LIN {X 0,Y 559.905,Z 784.141,A -85,B 0,C 180,E1 26458.055,E2 26458.055} C_VEL
LIN {X 0,Y 559.916,Z 781.549,A -85,B 0,C 180,E1 26456.109,E2 26456.109} C_VEL
LIN {X 0,Y 559.927,Z 777.44,A -85,B 0,C 180,E1 26454.261,E2 26454.261} C_VEL
LIN {X 0,Y 559.97,Z 771.528,A -85,B 0,C 180,E1 26452.407,E2 26452.407} C_VEL
LIN {X 0,Y 560.042,Z 763.726,A -85,B 0,C 180,E1 26450.546,E2 26450.546} C_VEL
LIN {X 0,Y 560.172,Z 754.398,A -85,B 0,C 180,E1 26448.781,E2 26448.781} C_VEL
LIN {X 0,Y 560.352,Z 743.578,A -85,B 0,C 180,E1 26447.112,E2 26447.112} C_VEL
LIN {X 0,Y 560.59,Z 731.187,A -85,B 0,C 180,E1 26445.54,E2 26445.54} C_VEL
LIN {X 0,Y 560.897,Z 717.221,A -85,B 0,C 180,E1 26444.066,E2 26444.066} C_VEL
LIN {X 0,Y 561.232,Z 702.873,A -85,B 0,C 180,E1 26442.798,E2 26442.798} C_VEL
LIN {X 0,Y 561.61,Z 686.59,A -85,B 0,C 180,E1 26441.61,E2 26441.61} C_VEL
LIN {X 0,Y 561.993,Z 668.948,A -85,B 0,C 180,E1 26440.567,E2 26440.567} C_VEL
LIN {X 0,Y 562.027,Z 667.326,A -85,B 0,C 180,E1 26440.483,E2 26440.483} C_VEL
LIN {X 0,Y 561.268,Z 660.484,A -85,B 0,C 180,E1 26440.115,E2 26440.115} C_VEL
LIN {X 0,Y 555.955,Z 643.327,A -85,B 0,C 180,E1 26439.189,E2 26439.189} C_VEL
LIN {X 0,Y 555.08,Z 636.153,A -85,B 0,C 180,E1 26438.903,E2 26438.903} C_VEL
LIN {X 0,Y 555.365,Z 617.419,A -85,B 0,C 180,E1 26438.404,E2 26438.404} C_VEL
LIN {X 0,Y 555.537,Z 595.534,A -85,B 0,C 180,E1 26438.046,E2 26438.046} C_VEL
LIN {X 0,Y 556.229,Z 411.604,A -85,B 0,C 180,E1 26435.545,E2 26435.545} C_VEL
LIN {X 0,Y 554.815,Z 403.726,A -85,B 0,C 180,E1 26435.342,E2 26435.342} C_VEL
LIN {X 0,Y 555.413,Z 371.536,A -85,B 0,C 180,E1 26432.441,E2 26432.441} C_VEL
LIN {X 0,Y 555.301,Z 368.267,A -85,B 0,C 180,E1 26432.139,E2 26432.139} C_VEL
LIN {X 0,Y 552.299,Z 358.003,A -85,B 0,C 180,E1 26431.014,E2 26431.014} C_VEL
LIN {X 0,Y 552.268,Z 358.001,A -85,B 0,C 180,E1 26427.718,E2 26427.718} C_VEL
LIN {X 0,Y 552.338,Z 357.999,A -85,B 0,C 180,E1 26424.549,E2 26424.549} C_VEL
LIN {X 0,Y 552.269,Z 358,A -85,B 0,C 180,E1 26421.346,E2 26421.346} C_VEL
LIN {X 0,Y 552.297,Z 358.001,A -85,B 0,C 180,E1 26418.079,E2 26418.079} C_VEL
LIN {X 0,Y 552.288,Z 357.999,A -85,B 0,C 180,E1 26414.938,E2 26414.938} C_VEL
LIN {X 0,Y 552.269,Z 357.999,A -85,B 0,C 180,E1 26411.607,E2 26411.607} C_VEL
LIN {X 0,Y 552.329,Z 357.999,A -85,B 0,C 180,E1 26408.516,E2 26408.516} C_VEL
LIN {X 0,Y 552.266,Z 358,A -85,B 0,C 180,E1 26405.262,E2 26405.262} C_VEL
LIN {X 0,Y 552.312,Z 358,A -85,B 0,C 180,E1 26402.034,E2 26402.034} C_VEL
LIN {X 0,Y 552.27,Z 357.999,A -85,B 0,C 180,E1 26399.02,E2 26399.02} C_VEL
LIN {X 0,Y 552.278,Z 358,A -85,B 0,C 180,E1 26395.631,E2 26395.631} C_VEL
LIN {X 0,Y 552.299,Z 357.998,A -85,B 0,C 180,E1 26392.569,E2 26392.569} C_VEL
LIN {X 0,Y 552.267,Z 358,A -85,B 0,C 180,E1 26389.349,E2 26389.349} C_VEL
LIN {X 0,Y 552.335,Z 357.998,A -85,B 0,C 180,E1 26386.187,E2 26386.187} C_VEL
LIN {X 0,Y 552.263,Z 357.998,A -85,B 0,C 180,E1 26383.08,E2 26383.08} C_VEL
LIN {X 0,Y 552.322,Z 357.999,A -85,B 0,C 180,E1 26379.903,E2 26379.903} C_VEL
LIN {X 0,Y 552.271,Z 357.999,A -85,B 0,C 180,E1 26376.758,E2 26376.758} C_VEL
LIN {X 0,Y 552.272,Z 357.999,A -85,B 0,C 180,E1 26373.321,E2 26373.321} C_VEL
LIN {X 0,Y 552.311,Z 357.999,A -85,B 0,C 180,E1 26370.207,E2 26370.207} C_VEL
LIN {X 0,Y 552.263,Z 357.998,A -85,B 0,C 180,E1 26366.99,E2 26366.99} C_VEL
LIN {X 0,Y 552.327,Z 357.999,A -85,B 0,C 180,E1 26363.764,E2 26363.764} C_VEL
LIN {X 0,Y 552.268,Z 357.999,A -85,B 0,C 180,E1 26360.622,E2 26360.622} C_VEL
LIN {X 0,Y 552.277,Z 358,A -85,B 0,C 180,E1 26357.24,E2 26357.24} C_VEL
LIN {X 0,Y 552.287,Z 358,A -85,B 0,C 180,E1 26354.243,E2 26354.243} C_VEL
LIN {X 0,Y 552.265,Z 358,A -85,B 0,C 180,E1 26350.921,E2 26350.921} C_VEL
LIN {X 0,Y 552.339,Z 357.999,A -85,B 0,C 180,E1 26347.769,E2 26347.769} C_VEL
LIN {X 0,Y 552.263,Z 358,A -85,B 0,C 180,E1 26344.59,E2 26344.59} C_VEL
LIN {X 0,Y 552.302,Z 358,A -85,B 0,C 180,E1 26341.331,E2 26341.331} C_VEL
LIN {X 0,Y 552.27,Z 358,A -85,B 0,C 180,E1 26338.312,E2 26338.312} C_VEL
LIN {X 0,Y 552.267,Z 358.001,A -85,B 0,C 180,E1 26334.849,E2 26334.849} C_VEL
LIN {X 0,Y 552.334,Z 358.001,A -85,B 0,C 180,E1 26331.613,E2 26331.613} C_VEL
LIN {X 0,Y 552.262,Z 358,A -85,B 0,C 180,E1 26328.394,E2 26328.394} C_VEL
LIN {X 0,Y 552.292,Z 358.001,A -85,B 0,C 180,E1 26325.085,E2 26325.085} C_VEL
LIN {X 0,Y 552.275,Z 358,A -85,B 0,C 180,E1 26322.057,E2 26322.057} C_VEL
LIN {X 0,Y 552.266,Z 358.001,A -85,B 0,C 180,E1 26318.654,E2 26318.654} C_VEL
LIN {X 0,Y 552.33,Z 358.001,A -85,B 0,C 180,E1 26315.45,E2 26315.45} C_VEL
LIN {X 0,Y 552.26,Z 358.003,A -85,B 0,C 180,E1 26312.274,E2 26312.274} C_VEL
LIN {X 0,Y 552.306,Z 358.003,A -85,B 0,C 180,E1 26309.024,E2 26309.024} C_VEL
LIN {X 0,Y 552.265,Z 358.028,A -85,B 0,C 180,E1 26308.41,E2 26308.41} C_VEL
LIN {X 0,Y 554.662,Z 367.675,A -85,B 0,C 180,E1 26307.134,E2 26307.134} C_VEL
LIN {X 0,Y 554.097,Z 397.179,A -85,B 0,C 180,E1 26303.728,E2 26303.728} C_VEL
LIN {X 0,Y 553.581,Z 425.304,A -85,B 0,C 180,E1 26300.512,E2 26300.512} C_VEL
LIN {X 0,Y 553.056,Z 456.362,A -85,B 0,C 180,E1 26297.03,E2 26297.03} C_VEL
LIN {X 0,Y 552.732,Z 481.06,A -85,B 0,C 180,E1 26294.338,E2 26294.338} C_VEL
LIN {X 0,Y 553.464,Z 488.754,A -85,B 0,C 180,E1 26294.218,E2 26294.218} C_VEL
LIN {X 0,Y 553.107,Z 591.575,A -85,B 0,C 180,E1 26292.854,E2 26292.854} C_VEL
LIN {X 0,Y 553.014,Z 606.185,A -85,B 0,C 180,E1 26292.489,E2 26292.489} C_VEL
LIN {X 0,Y 552.864,Z 619.873,A -85,B 0,C 180,E1 26291.946,E2 26291.946} C_VEL
LIN {X 0,Y 552.676,Z 631.744,A -85,B 0,C 180,E1 26291.319,E2 26291.319} C_VEL
LIN {X 0,Y 552.466,Z 644.76,A -85,B 0,C 180,E1 26290.427,E2 26290.427} C_VEL
LIN {X 0,Y 552.307,Z 655.904,A -85,B 0,C 180,E1 26289.43,E2 26289.43} C_VEL
LIN {X 0,Y 552.166,Z 665.819,A -85,B 0,C 180,E1 26288.33,E2 26288.33} C_VEL
LIN {X 0,Y 552.044,Z 675.086,A -85,B 0,C 180,E1 26287.003,E2 26287.003} C_VEL
LIN {X 0,Y 551.979,Z 681.519,A -85,B 0,C 180,E1 26285.822,E2 26285.822} C_VEL
LIN {X 0,Y 551.94,Z 687.227,A -85,B 0,C 180,E1 26284.468,E2 26284.468} C_VEL
LIN {X 0,Y 551.92,Z 691.681,A -85,B 0,C 180,E1 26282.908,E2 26282.908} C_VEL
LIN {X 0,Y 551.916,Z 693.98,A -85,B 0,C 180,E1 26281.557,E2 26281.557} C_VEL
LIN {X 0,Y 551.916,Z 694.996,A -85,B 0,C 180,E1 26280,E2 26280} C_VEL
LIN {X 0,Y 551.918,Z 694.092,A -85,B 0,C 180,E1 26278.443,E2 26278.443} C_VEL
LIN {X 0,Y 551.919,Z 691.869,A -85,B 0,C 180,E1 26277.093,E2 26277.093} C_VEL
LIN {X 0,Y 551.935,Z 687.911,A -85,B 0,C 180,E1 26275.637,E2 26275.637} C_VEL
LIN {X 0,Y 551.974,Z 681.957,A -85,B 0,C 180,E1 26274.178,E2 26274.178} C_VEL
LIN {X 0,Y 552.043,Z 675.194,A -85,B 0,C 180,E1 26272.926,E2 26272.926} C_VEL
LIN {X 0,Y 552.158,Z 666.551,A -85,B 0,C 180,E1 26271.671,E2 26271.671} C_VEL
LIN {X 0,Y 552.296,Z 656.805,A -85,B 0,C 180,E1 26270.57,E2 26270.57} C_VEL
LIN {X 0,Y 552.442,Z 647.08,A -85,B 0,C 180,E1 26269.678,E2 26269.678} C_VEL
LIN {X 0,Y 552.635,Z 634.983,A -85,B 0,C 180,E1 26268.785,E2 26268.785} C_VEL
LIN {X 0,Y 552.84,Z 621.669,A -85,B 0,C 180,E1 26268.049,E2 26268.049} C_VEL
LIN {X 0,Y 552.988,Z 609.624,A -85,B 0,C 180,E1 26267.546,E2 26267.546} C_VEL
LIN {X 0,Y 553.147,Z 595.043,A -85,B 0,C 180,E1 26267.121,E2 26267.121} C_VEL
LIN {X 0,Y 553.225,Z 571.612,A -85,B 0,C 180,E1 26266.771,E2 26266.771} C_VEL
LIN {X 0,Y 553.235,Z 484.541,A -85,B 0,C 180,E1 26265.631,E2 26265.631} C_VEL
LIN {X 0,Y 552.731,Z 480.548,A -85,B 0,C 180,E1 26265.544,E2 26265.544} C_VEL
LIN {X 0,Y 553.202,Z 451.312,A -85,B 0,C 180,E1 26262.271,E2 26262.271} C_VEL
LIN {X 0,Y 553.876,Z 420.903,A -85,B 0,C 180,E1 26258.781,E2 26258.781} C_VEL
LIN {X 0,Y 554.628,Z 391.683,A -85,B 0,C 180,E1 26255.39,E2 26255.39} C_VEL
LIN {X 0,Y 555.131,Z 368.311,A -85,B 0,C 180,E1 26252.618,E2 26252.618} C_VEL
LIN {X 0,Y 552.283,Z 358.006,A -85,B 0,C 180,E1 26251.153,E2 26251.153} C_VEL
LIN {X 0,Y 552.267,Z 358.004,A -85,B 0,C 180,E1 26247.841,E2 26247.841} C_VEL
LIN {X 0,Y 552.323,Z 358.001,A -85,B 0,C 180,E1 26244.727,E2 26244.727} C_VEL
LIN {X 0,Y 552.263,Z 358.003,A -85,B 0,C 180,E1 26241.611,E2 26241.611} C_VEL
LIN {X 0,Y 552.335,Z 358,A -85,B 0,C 180,E1 26238.506,E2 26238.506} C_VEL
LIN {X 0,Y 552.264,Z 358.002,A -85,B 0,C 180,E1 26235.359,E2 26235.359} C_VEL
LIN {X 0,Y 552.301,Z 358.003,A -85,B 0,C 180,E1 26232.077,E2 26232.077} C_VEL
LIN {X 0,Y 552.274,Z 358.002,A -85,B 0,C 180,E1 26229.043,E2 26229.043} C_VEL
LIN {X 0,Y 552.27,Z 358.005,A -85,B 0,C 180,E1 26225.621,E2 26225.621} C_VEL
LIN {X 0,Y 552.346,Z 358.153,A -85,B 0,C 180,E1 26222.461,E2 26222.461} C_VEL
LIN {X 0,Y 556.828,Z 371.461,A -85,B 0,C 180,E1 26221.141,E2 26221.141} C_VEL
LIN {X 0,Y 556.025,Z 413.458,A -85,B 0,C 180,E1 26218.049,E2 26218.049} C_VEL
LIN {X 0,Y 555.335,Z 457.917,A -85,B 0,C 180,E1 26214.917,E2 26214.917} C_VEL
LIN {X 0,Y 555.345,Z 463.245,A -85,B 0,C 180,E1 26214.568,E2 26214.568} C_VEL
LIN {X 0,Y 556.414,Z 472.063,A -85,B 0,C 180,E1 26214.395,E2 26214.395} C_VEL
LIN {X 0,Y 555.439,Z 672.312,A -85,B 0,C 180,E1 26211.656,E2 26211.656} C_VEL
LIN {X 0,Y 555.177,Z 691.233,A -85,B 0,C 180,E1 26211.202,E2 26211.202} C_VEL
LIN {X 0,Y 554.831,Z 709.39,A -85,B 0,C 180,E1 26210.574,E2 26210.574} C_VEL
LIN {X 0,Y 554.427,Z 727.031,A -85,B 0,C 180,E1 26209.764,E2 26209.764} C_VEL
LIN {X 0,Y 554.003,Z 743.688,A -85,B 0,C 180,E1 26208.799,E2 26208.799} C_VEL
LIN {X 0,Y 553.575,Z 759.623,A -85,B 0,C 180,E1 26207.664,E2 26207.664} C_VEL
LIN {X 0,Y 553.162,Z 774.553,A -85,B 0,C 180,E1 26206.378,E2 26206.378} C_VEL
LIN {X 0,Y 552.809,Z 788.017,A -85,B 0,C 180,E1 26204.99,E2 26204.99} C_VEL
LIN {X 0,Y 552.497,Z 800.914,A -85,B 0,C 180,E1 26203.394,E2 26203.394} C_VEL
LIN {X 0,Y 552.266,Z 812.229,A -85,B 0,C 180,E1 26201.699,E2 26201.699} C_VEL
LIN {X 0,Y 552.096,Z 822.169,A -85,B 0,C 180,E1 26199.871,E2 26199.871} C_VEL
LIN {X 0,Y 551.99,Z 830.178,A -85,B 0,C 180,E1 26198.018,E2 26198.018} C_VEL
LIN {X 0,Y 551.941,Z 836.414,A -85,B 0,C 180,E1 26196.136,E2 26196.136} C_VEL
LIN {X 0,Y 551.914,Z 840.877,A -85,B 0,C 180,E1 26194.26,E2 26194.26} C_VEL
LIN {X 0,Y 551.911,Z 843.792,A -85,B 0,C 180,E1 26192.284,E2 26192.284} C_VEL
LIN {X 0,Y 551.908,Z 844.94,A -85,B 0,C 180,E1 26190.311,E2 26190.311} C_VEL
LIN {X 0,Y 551.913,Z 844.416,A -85,B 0,C 180,E1 26188.443,E2 26188.443} C_VEL
LIN {X 0,Y 551.91,Z 842.163,A -85,B 0,C 180,E1 26186.469,E2 26186.469} C_VEL
LIN {X 0,Y 551.93,Z 838.35,A -85,B 0,C 180,E1 26184.595,E2 26184.595} C_VEL
LIN {X 0,Y 551.973,Z 832.818,A -85,B 0,C 180,E1 26182.715,E2 26182.715} C_VEL
LIN {X 0,Y 552.055,Z 825.427,A -85,B 0,C 180,E1 26180.829,E2 26180.829} C_VEL
LIN {X 0,Y 552.183,Z 816.517,A -85,B 0,C 180,E1 26179.04,E2 26179.04} C_VEL
LIN {X 0,Y 552.389,Z 805.985,A -85,B 0,C 180,E1 26177.323,E2 26177.323} C_VEL
LIN {X 0,Y 552.656,Z 794.351,A -85,B 0,C 180,E1 26175.756,E2 26175.756} C_VEL
LIN {X 0,Y 553.008,Z 780.575,A -85,B 0,C 180,E1 26174.21,E2 26174.21} C_VEL
LIN {X 0,Y 553.415,Z 765.602,A -85,B 0,C 180,E1 26172.819,E2 26172.819} C_VEL
LIN {X 0,Y 553.854,Z 749.432,A -85,B 0,C 180,E1 26171.583,E2 26171.583} C_VEL
LIN {X 0,Y 554.274,Z 733.051,A -85,B 0,C 180,E1 26170.56,E2 26170.56} C_VEL
LIN {X 0,Y 554.689,Z 715.808,A -85,B 0,C 180,E1 26169.696,E2 26169.696} C_VEL
LIN {X 0,Y 555.062,Z 697.521,A -85,B 0,C 180,E1 26168.994,E2 26168.994} C_VEL
LIN {X 0,Y 555.352,Z 678.843,A -85,B 0,C 180,E1 26168.48,E2 26168.48} C_VEL
LIN {X 0,Y 555.535,Z 658.475,A -85,B 0,C 180,E1 26168.131,E2 26168.131} C_VEL
LIN {X 0,Y 556.263,Z 469.166,A -85,B 0,C 180,E1 26165.558,E2 26165.558} C_VEL
LIN {X 0,Y 555.257,Z 462.604,A -85,B 0,C 180,E1 26165.417,E2 26165.417} C_VEL
LIN {X 0,Y 556.077,Z 416.365,A -85,B 0,C 180,E1 26162.128,E2 26162.128} C_VEL
LIN {X 0,Y 556.788,Z 373.888,A -85,B 0,C 180,E1 26159.037,E2 26159.037} C_VEL
LIN {X 0,Y 556.714,Z 371.068,A -85,B 0,C 180,E1 26158.815,E2 26158.815} C_VEL
LIN {X 0,Y 552.323,Z 357.992,A -85,B 0,C 180,E1 26157.521,E2 26157.521} C_VEL
LIN {X 0,Y 552.27,Z 358.001,A -85,B 0,C 180,E1 26154.38,E2 26154.38} C_VEL
LIN {X 0,Y 552.273,Z 358.001,A -85,B 0,C 180,E1 26150.947,E2 26150.947} C_VEL
LIN {X 0,Y 552.3,Z 358.002,A -85,B 0,C 180,E1 26147.923,E2 26147.923} C_VEL
LIN {X 0,Y 552.263,Z 358.001,A -85,B 0,C 180,E1 26144.641,E2 26144.641} C_VEL
LIN {X 0,Y 552.338,Z 358,A -85,B 0,C 180,E1 26141.458,E2 26141.458} C_VEL
LIN {X 0,Y 552.262,Z 358.002,A -85,B 0,C 180,E1 26138.377,E2 26138.377} C_VEL
LIN {X 0,Y 552.307,Z 358.003,A -85,B 0,C 180,E1 26135.148,E2 26135.148} C_VEL
LIN {X 0,Y 552.271,Z 358.005,A -85,B 0,C 180,E1 26132.037,E2 26132.037} C_VEL
LIN {X 0,Y 552.288,Z 358.066,A -85,B 0,C 180,E1 26128.808,E2 26128.808} C_VEL
LIN {X 0,Y 555.368,Z 369.2,A -85,B 0,C 180,E1 26127.652,E2 26127.652} C_VEL
LIN {X 0,Y 555.188,Z 387.302,A -85,B 0,C 180,E1 26126.067,E2 26126.067} C_VEL
LIN {X 0,Y 554.885,Z 404.57,A -85,B 0,C 180,E1 26124.525,E2 26124.525} C_VEL
LIN {X 0,Y 556.376,Z 413.773,A -85,B 0,C 180,E1 26124.328,E2 26124.328} C_VEL
LIN {X 0,Y 555.435,Z 612.55,A -85,B 0,C 180,E1 26121.607,E2 26121.607} C_VEL
LIN {X 0,Y 555.154,Z 632.028,A -85,B 0,C 180,E1 26121.134,E2 26121.134} C_VEL
LIN {X 0,Y 554.826,Z 649.668,A -85,B 0,C 180,E1 26120.518,E2 26120.518} C_VEL
LIN {X 0,Y 554.401,Z 668.293,A -85,B 0,C 180,E1 26119.655,E2 26119.655} C_VEL
LIN {X 0,Y 553.957,Z 685.572,A -85,B 0,C 180,E1 26118.63,E2 26118.63} C_VEL
LIN {X 0,Y 553.523,Z 701.786,A -85,B 0,C 180,E1 26117.449,E2 26117.449} C_VEL
LIN {X 0,Y 553.108,Z 716.635,A -85,B 0,C 180,E1 26116.13,E2 26116.13} C_VEL
LIN {X 0,Y 552.756,Z 730.434,A -85,B 0,C 180,E1 26114.669,E2 26114.669} C_VEL
LIN {X 0,Y 552.461,Z 742.929,A -85,B 0,C 180,E1 26113.075,E2 26113.075} C_VEL
LIN {X 0,Y 552.229,Z 753.85,A -85,B 0,C 180,E1 26111.382,E2 26111.382} C_VEL
LIN {X 0,Y 552.076,Z 763.297,A -85,B 0,C 180,E1 26109.591,E2 26109.591} C_VEL
LIN {X 0,Y 551.989,Z 771.211,A -85,B 0,C 180,E1 26107.703,E2 26107.703} C_VEL
LIN {X 0,Y 551.94,Z 777.184,A -85,B 0,C 180,E1 26105.822,E2 26105.822} C_VEL
LIN {X 0,Y 551.916,Z 781.378,A -85,B 0,C 180,E1 26103.947,E2 26103.947} C_VEL
LIN {X 0,Y 551.91,Z 784.066,A -85,B 0,C 180,E1 26101.972,E2 26101.972} C_VEL
LIN {X 0,Y 551.914,Z 784.996,A -85,B 0,C 180,E1 26100,E2 26100} C_VEL
LIN {X 0,Y 551.905,Z 784.136,A -85,B 0,C 180,E1 26098.027,E2 26098.027} C_VEL
LIN {X 0,Y 551.916,Z 781.543,A -85,B 0,C 180,E1 26096.052,E2 26096.052} C_VEL
LIN {X 0,Y 551.931,Z 777.438,A -85,B 0,C 180,E1 26094.177,E2 26094.177} C_VEL
LIN {X 0,Y 551.983,Z 771.52,A -85,B 0,C 180,E1 26092.297,E2 26092.297} C_VEL
LIN {X 0,Y 552.067,Z 763.716,A -85,B 0,C 180,E1 26090.408,E2 26090.408} C_VEL
LIN {X 0,Y 552.223,Z 754.391,A -85,B 0,C 180,E1 26088.617,E2 26088.617} C_VEL
LIN {X 0,Y 552.445,Z 743.572,A -85,B 0,C 180,E1 26086.924,E2 26086.924} C_VEL
LIN {X 0,Y 552.729,Z 731.174,A -85,B 0,C 180,E1 26085.33,E2 26085.33} C_VEL
LIN {X 0,Y 553.092,Z 717.211,A -85,B 0,C 180,E1 26083.835,E2 26083.835} C_VEL
LIN {X 0,Y 553.501,Z 702.448,A -85,B 0,C 180,E1 26082.516,E2 26082.516} C_VEL
LIN {X 0,Y 553.925,Z 686.915,A -85,B 0,C 180,E1 26081.368,E2 26081.368} C_VEL
LIN {X 0,Y 554.387,Z 668.945,A -85,B 0,C 180,E1 26080.29,E2 26080.29} C_VEL
LIN {X 0,Y 554.812,Z 650.474,A -85,B 0,C 180,E1 26079.426,E2 26079.426} C_VEL
LIN {X 0,Y 555.08,Z 636.153,A -85,B 0,C 180,E1 26078.903,E2 26078.903} C_VEL
LIN {X 0,Y 554.251,Z 628.853,A -85,B 0,C 180,E1 26078.64,E2 26078.64} C_VEL
LIN {X 0,Y 549.168,Z 611.542,A -85,B 0,C 180,E1 26078.024,E2 26078.024} C_VEL
LIN {X 0,Y 548.1,Z 604.053,A -85,B 0,C 180,E1 26077.853,E2 26077.853} C_VEL
LIN {X 0,Y 548.08,Z 602.958,A -85,B 0,C 180,E1 26077.836,E2 26077.836} C_VEL
LIN {X 0,Y 548.93,Z 412.864,A -85,B 0,C 180,E1 26075.221,E2 26075.221} C_VEL
LIN {X 0,Y 547.312,Z 404.139,A -85,B 0,C 180,E1 26075.007,E2 26075.007} C_VEL
LIN {X 0,Y 547.955,Z 374.089,A -85,B 0,C 180,E1 26072.27,E2 26072.27} C_VEL
LIN {X 0,Y 547.873,Z 370.936,A -85,B 0,C 180,E1 26071.976,E2 26071.976} C_VEL
LIN {X 0,Y 544.397,Z 358.989,A -85,B 0,C 180,E1 26070.667,E2 26070.667} C_VEL
LIN {X 0,Y 544.329,Z 358.99,A -85,B 0,C 180,E1 26067.439,E2 26067.439} C_VEL
LIN {X 0,Y 544.354,Z 358.991,A -85,B 0,C 180,E1 26064.098,E2 26064.098} C_VEL
LIN {X 0,Y 544.354,Z 358.989,A -85,B 0,C 180,E1 26060.948,E2 26060.948} C_VEL
LIN {X 0,Y 544.329,Z 358.989,A -85,B 0,C 180,E1 26057.613,E2 26057.613} C_VEL
LIN {X 0,Y 544.397,Z 358.989,A -85,B 0,C 180,E1 26054.401,E2 26054.401} C_VEL
LIN {X 0,Y 544.335,Z 358.988,A -85,B 0,C 180,E1 26051.117,E2 26051.117} C_VEL
LIN {X 0,Y 544.334,Z 358.989,A -85,B 0,C 180,E1 26047.657,E2 26047.657} C_VEL
LIN {X 0,Y 544.387,Z 358.989,A -85,B 0,C 180,E1 26044.445,E2 26044.445} C_VEL
LIN {X 0,Y 544.328,Z 358.989,A -85,B 0,C 180,E1 26041.198,E2 26041.198} C_VEL
LIN {X 0,Y 544.365,Z 358.989,A -85,B 0,C 180,E1 26037.929,E2 26037.929} C_VEL
LIN {X 0,Y 544.345,Z 358.988,A -85,B 0,C 180,E1 26034.759,E2 26034.759} C_VEL
LIN {X 0,Y 544.332,Z 358.988,A -85,B 0,C 180,E1 26031.441,E2 26031.441} C_VEL
LIN {X 0,Y 544.393,Z 358.989,A -85,B 0,C 180,E1 26028.194,E2 26028.194} C_VEL
LIN {X 0,Y 544.328,Z 358.989,A -85,B 0,C 180,E1 26024.94,E2 26024.94} C_VEL
LIN {X 0,Y 544.353,Z 358.989,A -85,B 0,C 180,E1 26021.657,E2 26021.657} C_VEL
LIN {X 0,Y 544.346,Z 358.987,A -85,B 0,C 180,E1 26018.556,E2 26018.556} C_VEL
LIN {X 0,Y 544.33,Z 358.988,A -85,B 0,C 180,E1 26015.27,E2 26015.27} C_VEL
LIN {X 0,Y 544.395,Z 358.988,A -85,B 0,C 180,E1 26012,E2 26012} C_VEL
LIN {X 0,Y 544.325,Z 358.987,A -85,B 0,C 180,E1 26008.842,E2 26008.842} C_VEL
LIN {X 0,Y 544.36,Z 358.989,A -85,B 0,C 180,E1 26005.576,E2 26005.576} C_VEL
LIN {X 0,Y 544.337,Z 358.987,A -85,B 0,C 180,E1 26002.506,E2 26002.506} C_VEL
LIN {X 0,Y 544.329,Z 358.989,A -85,B 0,C 180,E1 25999.094,E2 25999.094} C_VEL
LIN {X 0,Y 544.399,Z 358.988,A -85,B 0,C 180,E1 25995.861,E2 25995.861} C_VEL
LIN {X 0,Y 544.327,Z 358.988,A -85,B 0,C 180,E1 25992.578,E2 25992.578} C_VEL
LIN {X 0,Y 544.343,Z 358.989,A -85,B 0,C 180,E1 25989.219,E2 25989.219} C_VEL
LIN {X 0,Y 544.348,Z 358.988,A -85,B 0,C 180,E1 25986.165,E2 25986.165} C_VEL
LIN {X 0,Y 544.327,Z 358.989,A -85,B 0,C 180,E1 25982.9,E2 25982.9} C_VEL
LIN {X 0,Y 544.383,Z 358.988,A -85,B 0,C 180,E1 25979.784,E2 25979.784} C_VEL
LIN {X 0,Y 544.322,Z 358.99,A -85,B 0,C 180,E1 25976.56,E2 25976.56} C_VEL
LIN {X 0,Y 544.374,Z 358.991,A -85,B 0,C 180,E1 25973.349,E2 25973.349} C_VEL
LIN {X 0,Y 544.328,Z 358.99,A -85,B 0,C 180,E1 25970.265,E2 25970.265} C_VEL
LIN {X 0,Y 544.331,Z 358.989,A -85,B 0,C 180,E1 25966.822,E2 25966.822} C_VEL
LIN {X 0,Y 544.378,Z 358.989,A -85,B 0,C 180,E1 25963.642,E2 25963.642} C_VEL
LIN {X 0,Y 544.322,Z 358.99,A -85,B 0,C 180,E1 25960.423,E2 25960.423} C_VEL
LIN {X 0,Y 544.373,Z 358.991,A -85,B 0,C 180,E1 25957.177,E2 25957.177} C_VEL
LIN {X 0,Y 544.329,Z 358.991,A -85,B 0,C 180,E1 25954.062,E2 25954.062} C_VEL
LIN {X 0,Y 544.327,Z 358.993,A -85,B 0,C 180,E1 25950.585,E2 25950.585} C_VEL
LIN {X 0,Y 544.347,Z 359.064,A -85,B 0,C 180,E1 25948.737,E2 25948.737} C_VEL
LIN {X 0,Y 547.079,Z 370.15,A -85,B 0,C 180,E1 25947.247,E2 25947.247} C_VEL
LIN {X 0,Y 546.417,Z 399.154,A -85,B 0,C 180,E1 25943.853,E2 25943.853} C_VEL
LIN {X 0,Y 545.833,Z 427.365,A -85,B 0,C 180,E1 25940.592,E2 25940.592} C_VEL
LIN {X 0,Y 545.231,Z 458.425,A -85,B 0,C 180,E1 25937.063,E2 25937.063} C_VEL
LIN {X 0,Y 544.885,Z 481.01,A -85,B 0,C 180,E1 25934.567,E2 25934.567} C_VEL
LIN {X 0,Y 545.738,Z 489.353,A -85,B 0,C 180,E1 25934.428,E2 25934.428} C_VEL
LIN {X 0,Y 545.31,Z 591.265,A -85,B 0,C 180,E1 25933.048,E2 25933.048} C_VEL
LIN {X 0,Y 545.199,Z 605.746,A -85,B 0,C 180,E1 25932.687,E2 25932.687} C_VEL
LIN {X 0,Y 545.041,Z 618.639,A -85,B 0,C 180,E1 25932.179,E2 25932.179} C_VEL
LIN {X 0,Y 544.846,Z 629.906,A -85,B 0,C 180,E1 25931.592,E2 25931.592} C_VEL
LIN {X 0,Y 544.627,Z 640.473,A -85,B 0,C 180,E1 25930.9,E2 25930.9} C_VEL
LIN {X 0,Y 544.455,Z 652.186,A -85,B 0,C 180,E1 25929.941,E2 25929.941} C_VEL
LIN {X 0,Y 544.266,Z 662.273,A -85,B 0,C 180,E1 25928.877,E2 25928.877} C_VEL
LIN {X 0,Y 544.131,Z 670.457,A -85,B 0,C 180,E1 25927.815,E2 25927.815} C_VEL
LIN {X 0,Y 544.028,Z 678.362,A -85,B 0,C 180,E1 25926.543,E2 25926.543} C_VEL
LIN {X 0,Y 543.957,Z 685.205,A -85,B 0,C 180,E1 25925.062,E2 25925.062} C_VEL
LIN {X 0,Y 543.927,Z 689.515,A -85,B 0,C 180,E1 25923.795,E2 25923.795} C_VEL
LIN {X 0,Y 543.918,Z 692.965,A -85,B 0,C 180,E1 25922.318,E2 25922.318} C_VEL
LIN {X 0,Y 543.918,Z 694.72,A -85,B 0,C 180,E1 25920.737,E2 25920.737} C_VEL
LIN {X 0,Y 543.916,Z 694.799,A -85,B 0,C 180,E1 25919.368,E2 25919.368} C_VEL
LIN {X 0,Y 543.918,Z 693.439,A -85,B 0,C 180,E1 25917.893,E2 25917.893} C_VEL
LIN {X 0,Y 543.928,Z 690.086,A -85,B 0,C 180,E1 25916.311,E2 25916.311} C_VEL
LIN {X 0,Y 543.951,Z 685.953,A -85,B 0,C 180,E1 25915.044,E2 25915.044} C_VEL
LIN {X 0,Y 544,Z 680.425,A -85,B 0,C 180,E1 25913.775,E2 25913.775} C_VEL
LIN {X 0,Y 544.105,Z 672.574,A -85,B 0,C 180,E1 25912.397,E2 25912.397} C_VEL
LIN {X 0,Y 544.235,Z 663.908,A -85,B 0,C 180,E1 25911.229,E2 25911.229} C_VEL
LIN {X 0,Y 544.403,Z 654.685,A -85,B 0,C 180,E1 25910.219,E2 25910.219} C_VEL
LIN {X 0,Y 544.605,Z 642.883,A -85,B 0,C 180,E1 25909.183,E2 25909.183} C_VEL
LIN {X 0,Y 544.817,Z 631.425,A -85,B 0,C 180,E1 25908.407,E2 25908.407} C_VEL
LIN {X 0,Y 545.009,Z 620.517,A -85,B 0,C 180,E1 25907.821,E2 25907.821} C_VEL
LIN {X 0,Y 545.203,Z 607.55,A -85,B 0,C 180,E1 25907.287,E2 25907.287} C_VEL
LIN {X 0,Y 545.355,Z 592.327,A -85,B 0,C 180,E1 25906.88,E2 25906.88} C_VEL
LIN {X 0,Y 545.533,Z 549.584,A -85,B 0,C 180,E1 25906.277,E2 25906.277} C_VEL
LIN {X 0,Y 545.601,Z 485.393,A -85,B 0,C 180,E1 25905.39,E2 25905.39} C_VEL
LIN {X 0,Y 544.938,Z 480.565,A -85,B 0,C 180,E1 25905.279,E2 25905.279} C_VEL
LIN {X 0,Y 545.605,Z 449.687,A -85,B 0,C 180,E1 25901.738,E2 25901.738} C_VEL
LIN {X 0,Y 546.305,Z 420.925,A -85,B 0,C 180,E1 25898.397,E2 25898.397} C_VEL
LIN {X 0,Y 547.149,Z 392.163,A -85,B 0,C 180,E1 25895.012,E2 25895.012} C_VEL
LIN {X 0,Y 547.774,Z 371.263,A -85,B 0,C 180,E1 25892.497,E2 25892.497} C_VEL
LIN {X 0,Y 544.393,Z 358.989,A -85,B 0,C 180,E1 25890.701,E2 25890.701} C_VEL
LIN {X 0,Y 544.325,Z 358.993,A -85,B 0,C 180,E1 25887.473,E2 25887.473} C_VEL
LIN {X 0,Y 544.35,Z 358.993,A -85,B 0,C 180,E1 25884.131,E2 25884.131} C_VEL
LIN {X 0,Y 544.341,Z 358.991,A -85,B 0,C 180,E1 25881.083,E2 25881.083} C_VEL
LIN {X 0,Y 544.331,Z 358.991,A -85,B 0,C 180,E1 25877.754,E2 25877.754} C_VEL
LIN {X 0,Y 544.39,Z 358.99,A -85,B 0,C 180,E1 25874.551,E2 25874.551} C_VEL
LIN {X 0,Y 544.327,Z 358.992,A -85,B 0,C 180,E1 25871.299,E2 25871.299} C_VEL
LIN {X 0,Y 544.36,Z 358.991,A -85,B 0,C 180,E1 25868.004,E2 25868.004} C_VEL
LIN {X 0,Y 544.337,Z 358.994,A -85,B 0,C 180,E1 25864.967,E2 25864.967} C_VEL
LIN {X 0,Y 544.356,Z 359.109,A -85,B 0,C 180,E1 25862.923,E2 25862.923} C_VEL
LIN {X 0,Y 549.483,Z 374.167,A -85,B 0,C 180,E1 25861.36,E2 25861.36} C_VEL
LIN {X 0,Y 548.631,Z 410.296,A -85,B 0,C 180,E1 25858.64,E2 25858.64} C_VEL
LIN {X 0,Y 547.839,Z 454.622,A -85,B 0,C 180,E1 25855.473,E2 25855.473} C_VEL
LIN {X 0,Y 547.789,Z 463.271,A -85,B 0,C 180,E1 25854.891,E2 25854.891} C_VEL
LIN {X 0,Y 549.074,Z 472.969,A -85,B 0,C 180,E1 25854.716,E2 25854.716} C_VEL
LIN {X 0,Y 548.002,Z 672.312,A -85,B 0,C 180,E1 25851.965,E2 25851.965} C_VEL
LIN {X 0,Y 547.699,Z 691.273,A -85,B 0,C 180,E1 25851.505,E2 25851.505} C_VEL
LIN {X 0,Y 547.304,Z 709.388,A -85,B 0,C 180,E1 25850.87,E2 25850.87} C_VEL
LIN {X 0,Y 546.837,Z 727.027,A -85,B 0,C 180,E1 25850.05,E2 25850.05} C_VEL
LIN {X 0,Y 546.332,Z 744.143,A -85,B 0,C 180,E1 25849.041,E2 25849.041} C_VEL
LIN {X 0,Y 545.831,Z 760.288,A -85,B 0,C 180,E1 25847.868,E2 25847.868} C_VEL
LIN {X 0,Y 545.34,Z 775.662,A -85,B 0,C 180,E1 25846.51,E2 25846.51} C_VEL
LIN {X 0,Y 544.914,Z 789.869,A -85,B 0,C 180,E1 25844.994,E2 25844.994} C_VEL
LIN {X 0,Y 544.563,Z 802.454,A -85,B 0,C 180,E1 25843.376,E2 25843.376} C_VEL
LIN {X 0,Y 544.302,Z 813.499,A -85,B 0,C 180,E1 25841.658,E2 25841.658} C_VEL
LIN {X 0,Y 544.117,Z 823.022,A -85,B 0,C 180,E1 25839.84,E2 25839.84} C_VEL
LIN {X 0,Y 544.001,Z 830.583,A -85,B 0,C 180,E1 25838.03,E2 25838.03} C_VEL
LIN {X 0,Y 543.945,Z 836.717,A -85,B 0,C 180,E1 25836.12,E2 25836.12} C_VEL
LIN {X 0,Y 543.915,Z 841.082,A -85,B 0,C 180,E1 25834.217,E2 25834.217} C_VEL
LIN {X 0,Y 543.911,Z 843.793,A -85,B 0,C 180,E1 25832.318,E2 25832.318} C_VEL
LIN {X 0,Y 543.908,Z 844.94,A -85,B 0,C 180,E1 25830.316,E2 25830.316} C_VEL
LIN {X 0,Y 543.912,Z 844.415,A -85,B 0,C 180,E1 25828.42,E2 25828.42} C_VEL
LIN {X 0,Y 543.911,Z 842.162,A -85,B 0,C 180,E1 25826.417,E2 25826.417} C_VEL
LIN {X 0,Y 543.932,Z 838.35,A -85,B 0,C 180,E1 25824.515,E2 25824.515} C_VEL
LIN {X 0,Y 543.981,Z 832.818,A -85,B 0,C 180,E1 25822.608,E2 25822.608} C_VEL
LIN {X 0,Y 544.081,Z 825.428,A -85,B 0,C 180,E1 25820.693,E2 25820.693} C_VEL
LIN {X 0,Y 544.234,Z 816.518,A -85,B 0,C 180,E1 25818.878,E2 25818.878} C_VEL
LIN {X 0,Y 544.468,Z 806.153,A -85,B 0,C 180,E1 25817.161,E2 25817.161} C_VEL
LIN {X 0,Y 544.781,Z 794.352,A -85,B 0,C 180,E1 25815.546,E2 25815.546} C_VEL
LIN {X 0,Y 545.178,Z 781.08,A -85,B 0,C 180,E1 25814.032,E2 25814.032} C_VEL
LIN {X 0,Y 545.649,Z 766.22,A -85,B 0,C 180,E1 25812.621,E2 25812.621} C_VEL
LIN {X 0,Y 546.159,Z 750.231,A -85,B 0,C 180,E1 25811.37,E2 25811.37} C_VEL
LIN {X 0,Y 546.667,Z 733.055,A -85,B 0,C 180,E1 25810.278,E2 25810.278} C_VEL
LIN {X 0,Y 547.139,Z 715.811,A -85,B 0,C 180,E1 25809.404,E2 25809.404} C_VEL
LIN {X 0,Y 547.566,Z 697.522,A -85,B 0,C 180,E1 25808.692,E2 25808.692} C_VEL
LIN {X 0,Y 547.901,Z 678.953,A -85,B 0,C 180,E1 25808.175,E2 25808.175} C_VEL
LIN {X 0,Y 548.111,Z 658.603,A -85,B 0,C 180,E1 25807.821,E2 25807.821} C_VEL
LIN {X 0,Y 548.942,Z 470.39,A -85,B 0,C 180,E1 25805.244,E2 25805.244} C_VEL
LIN {X 0,Y 547.752,Z 462.347,A -85,B 0,C 180,E1 25805.06,E2 25805.06} C_VEL
LIN {X 0,Y 548.687,Z 415.044,A -85,B 0,C 180,E1 25801.662,E2 25801.662} C_VEL
LIN {X 0,Y 549.502,Z 376.76,A -85,B 0,C 180,E1 25798.824,E2 25798.824} C_VEL
LIN {X 0,Y 549.418,Z 373.902,A -85,B 0,C 180,E1 25798.595,E2 25798.595} C_VEL
LIN {X 0,Y 544.34,Z 358.994,A -85,B 0,C 180,E1 25797.08,E2 25797.08} C_VEL
LIN {X 0,Y 544.375,Z 358.99,A -85,B 0,C 180,E1 25793.872,E2 25793.872} C_VEL
LIN {X 0,Y 544.325,Z 358.991,A -85,B 0,C 180,E1 25790.653,E2 25790.653} C_VEL
LIN {X 0,Y 544.386,Z 358.989,A -85,B 0,C 180,E1 25787.435,E2 25787.435} C_VEL
LIN {X 0,Y 544.331,Z 358.991,A -85,B 0,C 180,E1 25784.244,E2 25784.244} C_VEL
LIN {X 0,Y 544.333,Z 358.991,A -85,B 0,C 180,E1 25780.818,E2 25780.818} C_VEL
LIN {X 0,Y 544.356,Z 358.992,A -85,B 0,C 180,E1 25777.831,E2 25777.831} C_VEL
LIN {X 0,Y 544.325,Z 358.992,A -85,B 0,C 180,E1 25774.583,E2 25774.583} C_VEL
LIN {X 0,Y 544.393,Z 358.992,A -85,B 0,C 180,E1 25771.317,E2 25771.317} C_VEL
LIN {X 0,Y 544.391,Z 359.103,A -85,B 0,C 180,E1 25769.14,E2 25769.14} C_VEL
LIN {X 0,Y 547.942,Z 371.595,A -85,B 0,C 180,E1 25767.849,E2 25767.849} C_VEL
LIN {X 0,Y 547.681,Z 391.628,A -85,B 0,C 180,E1 25766.076,E2 25766.076} C_VEL
LIN {X 0,Y 547.428,Z 404.932,A -85,B 0,C 180,E1 25764.876,E2 25764.876} C_VEL
LIN {X 0,Y 549.047,Z 414.92,A -85,B 0,C 180,E1 25764.649,E2 25764.649} C_VEL
LIN {X 0,Y 547.998,Z 612.388,A -85,B 0,C 180,E1 25761.919,E2 25761.919} C_VEL
LIN {X 0,Y 547.685,Z 631.576,A -85,B 0,C 180,E1 25761.45,E2 25761.45} C_VEL
LIN {X 0,Y 547.309,Z 649.323,A -85,B 0,C 180,E1 25760.829,E2 25760.829} C_VEL
LIN {X 0,Y 546.807,Z 668.297,A -85,B 0,C 180,E1 25759.939,E2 25759.939} C_VEL
LIN {X 0,Y 546.295,Z 685.57,A -85,B 0,C 180,E1 25758.902,E2 25758.902} C_VEL
LIN {X 0,Y 545.792,Z 701.8,A -85,B 0,C 180,E1 25757.704,E2 25757.704} C_VEL
LIN {X 0,Y 545.306,Z 716.843,A -85,B 0,C 180,E1 25756.347,E2 25756.347} C_VEL
LIN {X 0,Y 544.9,Z 730.432,A -85,B 0,C 180,E1 25754.886,E2 25754.886} C_VEL
LIN {X 0,Y 544.556,Z 742.938,A -85,B 0,C 180,E1 25753.268,E2 25753.268} C_VEL
LIN {X 0,Y 544.287,Z 753.851,A -85,B 0,C 180,E1 25751.551,E2 25751.551} C_VEL
LIN {X 0,Y 544.11,Z 763.295,A -85,B 0,C 180,E1 25749.733,E2 25749.733} C_VEL
LIN {X 0,Y 543.999,Z 771.164,A -85,B 0,C 180,E1 25747.83,E2 25747.83} C_VEL
LIN {X 0,Y 543.944,Z 777.185,A -85,B 0,C 180,E1 25745.908,E2 25745.908} C_VEL
LIN {X 0,Y 543.915,Z 781.374,A -85,B 0,C 180,E1 25744.005,E2 25744.005} C_VEL
LIN {X 0,Y 543.91,Z 784.062,A -85,B 0,C 180,E1 25742.001,E2 25742.001} C_VEL
LIN {X 0,Y 543.914,Z 784.996,A -85,B 0,C 180,E1 25740,E2 25740} C_VEL
LIN {X 0,Y 543.905,Z 784.131,A -85,B 0,C 180,E1 25737.998,E2 25737.998} C_VEL
LIN {X 0,Y 543.917,Z 781.537,A -85,B 0,C 180,E1 25735.994,E2 25735.994} C_VEL
LIN {X 0,Y 543.936,Z 777.437,A -85,B 0,C 180,E1 25734.091,E2 25734.091} C_VEL
LIN {X 0,Y 543.993,Z 771.486,A -85,B 0,C 180,E1 25732.175,E2 25732.175} C_VEL
LIN {X 0,Y 544.098,Z 763.708,A -85,B 0,C 180,E1 25730.266,E2 25730.266} C_VEL
LIN {X 0,Y 544.279,Z 754.384,A -85,B 0,C 180,E1 25728.449,E2 25728.449} C_VEL
LIN {X 0,Y 544.55,Z 743.303,A -85,B 0,C 180,E1 25726.693,E2 25726.693} C_VEL
LIN {X 0,Y 544.876,Z 731.161,A -85,B 0,C 180,E1 25725.113,E2 25725.113} C_VEL
LIN {X 0,Y 545.295,Z 717.2,A -85,B 0,C 180,E1 25723.598,E2 25723.598} C_VEL
LIN {X 0,Y 545.757,Z 702.856,A -85,B 0,C 180,E1 25722.294,E2 25722.294} C_VEL
LIN {X 0,Y 546.26,Z 686.902,A -85,B 0,C 180,E1 25721.096,E2 25721.096} C_VEL
LIN {X 0,Y 546.794,Z 668.942,A -85,B 0,C 180,E1 25720.004,E2 25720.004} C_VEL
LIN {X 0,Y 547.283,Z 650.459,A -85,B 0,C 180,E1 25719.129,E2 25719.129} C_VEL
LIN {X 0,Y 547.671,Z 632.314,A -85,B 0,C 180,E1 25718.482,E2 25718.482} C_VEL
LIN {X 0,Y 547.994,Z 612.672,A -85,B 0,C 180,E1 25717.996,E2 25717.996} C_VEL
LIN {X 0,Y 548.08,Z 602.958,A -85,B 0,C 180,E1 25717.836,E2 25717.836} C_VEL
LIN {X 0,Y 547.196,Z 595.367,A -85,B 0,C 180,E1 25717.691,E2 25717.691} C_VEL
LIN {X 0,Y 541.437,Z 575.489,A -85,B 0,C 180,E1 25717.183,E2 25717.183} C_VEL
LIN {X 0,Y 540.767,Z 568.958,A -85,B 0,C 180,E1 25717.065,E2 25717.065} C_VEL
LIN {X 0,Y 541.609,Z 413.811,A -85,B 0,C 180,E1 25714.877,E2 25714.877} C_VEL
LIN {X 0,Y 539.869,Z 404.185,A -85,B 0,C 180,E1 25714.618,E2 25714.618} C_VEL
LIN {X 0,Y 540.554,Z 374.069,A -85,B 0,C 180,E1 25711.857,E2 25711.857} C_VEL
LIN {X 0,Y 536.427,Z 359.981,A -85,B 0,C 180,E1 25710.277,E2 25710.277} C_VEL
LIN {X 0,Y 536.405,Z 359.979,A -85,B 0,C 180,E1 25707.151,E2 25707.151} C_VEL
LIN {X 0,Y 536.394,Z 359.979,A -85,B 0,C 180,E1 25703.779,E2 25703.779} C_VEL
LIN {X 0,Y 536.465,Z 359.975,A -85,B 0,C 180,E1 25700.499,E2 25700.499} C_VEL
LIN {X 0,Y 536.393,Z 359.978,A -85,B 0,C 180,E1 25697.26,E2 25697.26} C_VEL
LIN {X 0,Y 536.403,Z 359.978,A -85,B 0,C 180,E1 25693.832,E2 25693.832} C_VEL
LIN {X 0,Y 536.445,Z 359.976,A -85,B 0,C 180,E1 25690.579,E2 25690.579} C_VEL
LIN {X 0,Y 536.39,Z 359.978,A -85,B 0,C 180,E1 25687.288,E2 25687.288} C_VEL
LIN {X 0,Y 536.421,Z 359.979,A -85,B 0,C 180,E1 25683.957,E2 25683.957} C_VEL
LIN {X 0,Y 536.412,Z 359.977,A -85,B 0,C 180,E1 25680.762,E2 25680.762} C_VEL
LIN {X 0,Y 536.39,Z 359.977,A -85,B 0,C 180,E1 25677.414,E2 25677.414} C_VEL
LIN {X 0,Y 536.457,Z 359.977,A -85,B 0,C 180,E1 25674.208,E2 25674.208} C_VEL
LIN {X 0,Y 536.391,Z 359.976,A -85,B 0,C 180,E1 25670.971,E2 25670.971} C_VEL
LIN {X 0,Y 536.403,Z 359.976,A -85,B 0,C 180,E1 25667.576,E2 25667.576} C_VEL
LIN {X 0,Y 536.434,Z 359.977,A -85,B 0,C 180,E1 25664.353,E2 25664.353} C_VEL
LIN {X 0,Y 536.387,Z 359.978,A -85,B 0,C 180,E1 25661.069,E2 25661.069} C_VEL
LIN {X 0,Y 536.436,Z 359.978,A -85,B 0,C 180,E1 25657.82,E2 25657.82} C_VEL
LIN {X 0,Y 536.4,Z 359.976,A -85,B 0,C 180,E1 25654.597,E2 25654.597} C_VEL
LIN {X 0,Y 536.388,Z 359.978,A -85,B 0,C 180,E1 25651.175,E2 25651.175} C_VEL
LIN {X 0,Y 536.453,Z 359.976,A -85,B 0,C 180,E1 25647.971,E2 25647.971} C_VEL
LIN {X 0,Y 536.387,Z 359.977,A -85,B 0,C 180,E1 25644.759,E2 25644.759} C_VEL
LIN {X 0,Y 536.411,Z 359.978,A -85,B 0,C 180,E1 25641.424,E2 25641.424} C_VEL
LIN {X 0,Y 536.412,Z 359.977,A -85,B 0,C 180,E1 25638.277,E2 25638.277} C_VEL
LIN {X 0,Y 536.389,Z 359.978,A -85,B 0,C 180,E1 25634.983,E2 25634.983} C_VEL
LIN {X 0,Y 536.453,Z 359.979,A -85,B 0,C 180,E1 25631.752,E2 25631.752} C_VEL
LIN {X 0,Y 536.391,Z 359.977,A -85,B 0,C 180,E1 25628.456,E2 25628.456} C_VEL
LIN {X 0,Y 536.391,Z 359.978,A -85,B 0,C 180,E1 25624.949,E2 25624.949} C_VEL
LIN {X 0,Y 536.451,Z 359.977,A -85,B 0,C 180,E1 25621.744,E2 25621.744} C_VEL
LIN {X 0,Y 536.385,Z 359.978,A -85,B 0,C 180,E1 25618.537,E2 25618.537} C_VEL
LIN {X 0,Y 536.418,Z 359.98,A -85,B 0,C 180,E1 25615.224,E2 25615.224} C_VEL
LIN {X 0,Y 536.404,Z 359.979,A -85,B 0,C 180,E1 25612.039,E2 25612.039} C_VEL
LIN {X 0,Y 536.387,Z 359.978,A -85,B 0,C 180,E1 25608.696,E2 25608.696} C_VEL
LIN {X 0,Y 536.451,Z 359.979,A -85,B 0,C 180,E1 25605.508,E2 25605.508} C_VEL
LIN {X 0,Y 536.386,Z 359.979,A -85,B 0,C 180,E1 25602.265,E2 25602.265} C_VEL
LIN {X 0,Y 536.404,Z 359.98,A -85,B 0,C 180,E1 25598.915,E2 25598.915} C_VEL
LIN {X 0,Y 536.409,Z 359.979,A -85,B 0,C 180,E1 25595.822,E2 25595.822} C_VEL
LIN {X 0,Y 536.384,Z 359.982,A -85,B 0,C 180,E1 25592.47,E2 25592.47} C_VEL
LIN {X 0,Y 536.454,Z 359.979,A -85,B 0,C 180,E1 25589.231,E2 25589.231} C_VEL
LIN {X 0,Y 536.466,Z 360.225,A -85,B 0,C 180,E1 25589.059,E2 25589.059} C_VEL
LIN {X 0,Y 539.498,Z 372.627,A -85,B 0,C 180,E1 25587.363,E2 25587.363} C_VEL
LIN {X 0,Y 538.752,Z 401.187,A -85,B 0,C 180,E1 25583.981,E2 25583.981} C_VEL
LIN {X 0,Y 538.09,Z 429.45,A -85,B 0,C 180,E1 25580.674,E2 25580.674} C_VEL
LIN {X 0,Y 537.43,Z 460.12,A -85,B 0,C 180,E1 25577.151,E2 25577.151} C_VEL
LIN {X 0,Y 537.068,Z 480.836,A -85,B 0,C 180,E1 25574.829,E2 25574.829} C_VEL
LIN {X 0,Y 538.06,Z 490.002,A -85,B 0,C 180,E1 25574.66,E2 25574.66} C_VEL
LIN {X 0,Y 537.568,Z 590.337,A -85,B 0,C 180,E1 25573.276,E2 25573.276} C_VEL
LIN {X 0,Y 537.45,Z 604.065,A -85,B 0,C 180,E1 25572.948,E2 25572.948} C_VEL
LIN {X 0,Y 537.276,Z 618.235,A -85,B 0,C 180,E1 25572.412,E2 25572.412} C_VEL
LIN {X 0,Y 537.035,Z 630.524,A -85,B 0,C 180,E1 25571.763,E2 25571.763} C_VEL
LIN {X 0,Y 536.786,Z 641.013,A -85,B 0,C 180,E1 25571.061,E2 25571.061} C_VEL
LIN {X 0,Y 536.574,Z 652.613,A -85,B 0,C 180,E1 25570.088,E2 25570.088} C_VEL
LIN {X 0,Y 536.346,Z 662.595,A -85,B 0,C 180,E1 25569.009,E2 25569.009} C_VEL
LIN {X 0,Y 536.179,Z 670.65,A -85,B 0,C 180,E1 25567.932,E2 25567.932} C_VEL
LIN {X 0,Y 536.048,Z 678.407,A -85,B 0,C 180,E1 25566.641,E2 25566.641} C_VEL
LIN {X 0,Y 535.964,Z 685.2,A -85,B 0,C 180,E1 25565.138,E2 25565.138} C_VEL
LIN {X 0,Y 535.929,Z 689.509,A -85,B 0,C 180,E1 25563.851,E2 25563.851} C_VEL
LIN {X 0,Y 535.919,Z 692.748,A -85,B 0,C 180,E1 25562.46,E2 25562.46} C_VEL
LIN {X 0,Y 535.917,Z 694.669,A -85,B 0,C 180,E1 25560.855,E2 25560.855} C_VEL
LIN {X 0,Y 535.916,Z 694.833,A -85,B 0,C 180,E1 25559.466,E2 25559.466} C_VEL
LIN {X 0,Y 535.916,Z 693.815,A -85,B 0,C 180,E1 25558.183,E2 25558.183} C_VEL
LIN {X 0,Y 535.925,Z 691.2,A -85,B 0,C 180,E1 25556.685,E2 25556.685} C_VEL
LIN {X 0,Y 535.95,Z 686.75,A -85,B 0,C 180,E1 25555.184,E2 25555.184} C_VEL
LIN {X 0,Y 536.004,Z 681.287,A -85,B 0,C 180,E1 25553.859,E2 25553.859} C_VEL
LIN {X 0,Y 536.114,Z 674.769,A -85,B 0,C 180,E1 25552.606,E2 25552.606} C_VEL
LIN {X 0,Y 536.292,Z 666.078,A -85,B 0,C 180,E1 25551.314,E2 25551.314} C_VEL
LIN {X 0,Y 536.497,Z 656.853,A -85,B 0,C 180,E1 25550.236,E2 25550.236} C_VEL
LIN {X 0,Y 536.73,Z 646.593,A -85,B 0,C 180,E1 25549.264,E2 25549.264} C_VEL
LIN {X 0,Y 537.024,Z 633.323,A -85,B 0,C 180,E1 25548.291,E2 25548.291} C_VEL
LIN {X 0,Y 537.264,Z 621.706,A -85,B 0,C 180,E1 25547.642,E2 25547.642} C_VEL
LIN {X 0,Y 537.476,Z 608.945,A -85,B 0,C 180,E1 25547.101,E2 25547.101} C_VEL
LIN {X 0,Y 537.652,Z 593.083,A -85,B 0,C 180,E1 25546.661,E2 25546.661} C_VEL
LIN {X 0,Y 537.864,Z 551.422,A -85,B 0,C 180,E1 25546.057,E2 25546.057} C_VEL
LIN {X 0,Y 538.145,Z 486.295,A -85,B 0,C 180,E1 25545.094,E2 25545.094} C_VEL
LIN {X 0,Y 537.233,Z 480.444,A -85,B 0,C 180,E1 25544.947,E2 25544.947} C_VEL
LIN {X 0,Y 537.955,Z 450.447,A -85,B 0,C 180,E1 25541.469,E2 25541.469} C_VEL
LIN {X 0,Y 538.738,Z 421.759,A -85,B 0,C 180,E1 25538.097,E2 25538.097} C_VEL
LIN {X 0,Y 539.705,Z 393.079,A -85,B 0,C 180,E1 25534.662,E2 25534.662} C_VEL
LIN {X 0,Y 540.389,Z 373.98,A -85,B 0,C 180,E1 25532.328,E2 25532.328} C_VEL
LIN {X 0,Y 536.413,Z 359.983,A -85,B 0,C 180,E1 25530.215,E2 25530.215} C_VEL
LIN {X 0,Y 536.401,Z 359.982,A -85,B 0,C 180,E1 25527.151,E2 25527.151} C_VEL
LIN {X 0,Y 536.39,Z 359.982,A -85,B 0,C 180,E1 25523.779,E2 25523.779} C_VEL
LIN {X 0,Y 536.462,Z 359.977,A -85,B 0,C 180,E1 25520.5,E2 25520.5} C_VEL
LIN {X 0,Y 536.39,Z 359.98,A -85,B 0,C 180,E1 25517.26,E2 25517.26} C_VEL
LIN {X 0,Y 536.401,Z 359.981,A -85,B 0,C 180,E1 25513.832,E2 25513.832} C_VEL
LIN {X 0,Y 536.444,Z 359.979,A -85,B 0,C 180,E1 25510.579,E2 25510.579} C_VEL
LIN {X 0,Y 536.388,Z 359.982,A -85,B 0,C 180,E1 25507.288,E2 25507.288} C_VEL
LIN {X 0,Y 536.421,Z 359.982,A -85,B 0,C 180,E1 25503.957,E2 25503.957} C_VEL
LIN {X 0,Y 536.398,Z 360.048,A -85,B 0,C 180,E1 25503.423,E2 25503.423} C_VEL
LIN {X 0,Y 542.203,Z 377.021,A -85,B 0,C 180,E1 25501.575,E2 25501.575} C_VEL
LIN {X 0,Y 541.104,Z 414.26,A -85,B 0,C 180,E1 25498.714,E2 25498.714} C_VEL
LIN {X 0,Y 540.157,Z 458.569,A -85,B 0,C 180,E1 25495.497,E2 25495.497} C_VEL
LIN {X 0,Y 540.143,Z 463.622,A -85,B 0,C 180,E1 25495.164,E2 25495.164} C_VEL
LIN {X 0,Y 541.481,Z 473.996,A -85,B 0,C 180,E1 25494.97,E2 25494.97} C_VEL
LIN {X 0,Y 540.582,Z 671.854,A -85,B 0,C 180,E1 25492.289,E2 25492.289} C_VEL
LIN {X 0,Y 540.251,Z 690.814,A -85,B 0,C 180,E1 25491.831,E2 25491.831} C_VEL
LIN {X 0,Y 539.792,Z 709.385,A -85,B 0,C 180,E1 25491.174,E2 25491.174} C_VEL
LIN {X 0,Y 539.261,Z 727.023,A -85,B 0,C 180,E1 25490.344,E2 25490.344} C_VEL
LIN {X 0,Y 538.703,Z 743.757,A -85,B 0,C 180,E1 25489.348,E2 25489.348} C_VEL
LIN {X 0,Y 538.147,Z 759.617,A -85,B 0,C 180,E1 25488.188,E2 25488.188} C_VEL
LIN {X 0,Y 537.604,Z 774.549,A -85,B 0,C 180,E1 25486.866,E2 25486.866} C_VEL
LIN {X 0,Y 537.13,Z 788.016,A -85,B 0,C 180,E1 25485.438,E2 25485.438} C_VEL
LIN {X 0,Y 536.712,Z 800.912,A -85,B 0,C 180,E1 25483.795,E2 25483.795} C_VEL
LIN {X 0,Y 536.395,Z 812.228,A -85,B 0,C 180,E1 25482.05,E2 25482.05} C_VEL
LIN {X 0,Y 536.164,Z 821.992,A -85,B 0,C 180,E1 25480.204,E2 25480.204} C_VEL
LIN {X 0,Y 536.025,Z 830.178,A -85,B 0,C 180,E1 25478.258,E2 25478.258} C_VEL
LIN {X 0,Y 535.949,Z 836.415,A -85,B 0,C 180,E1 25476.319,E2 25476.319} C_VEL
LIN {X 0,Y 535.917,Z 840.877,A -85,B 0,C 180,E1 25474.387,E2 25474.387} C_VEL
LIN {X 0,Y 535.911,Z 843.793,A -85,B 0,C 180,E1 25472.352,E2 25472.352} C_VEL
LIN {X 0,Y 535.908,Z 844.94,A -85,B 0,C 180,E1 25470.321,E2 25470.321} C_VEL
LIN {X 0,Y 535.911,Z 844.415,A -85,B 0,C 180,E1 25468.396,E2 25468.396} C_VEL
LIN {X 0,Y 535.913,Z 842.162,A -85,B 0,C 180,E1 25466.363,E2 25466.363} C_VEL
LIN {X 0,Y 535.934,Z 838.349,A -85,B 0,C 180,E1 25464.433,E2 25464.433} C_VEL
LIN {X 0,Y 535.992,Z 832.818,A -85,B 0,C 180,E1 25462.497,E2 25462.497} C_VEL
LIN {X 0,Y 536.107,Z 825.427,A -85,B 0,C 180,E1 25460.554,E2 25460.554} C_VEL
LIN {X 0,Y 536.289,Z 816.518,A -85,B 0,C 180,E1 25458.711,E2 25458.711} C_VEL
LIN {X 0,Y 536.558,Z 806.153,A -85,B 0,C 180,E1 25456.969,E2 25456.969} C_VEL
LIN {X 0,Y 536.917,Z 794.352,A -85,B 0,C 180,E1 25455.329,E2 25455.329} C_VEL
LIN {X 0,Y 537.394,Z 780.681,A -85,B 0,C 180,E1 25453.751,E2 25453.751} C_VEL
LIN {X 0,Y 537.942,Z 765.603,A -85,B 0,C 180,E1 25452.308,E2 25452.308} C_VEL
LIN {X 0,Y 538.522,Z 749.438,A -85,B 0,C 180,E1 25451.039,E2 25451.039} C_VEL
LIN {X 0,Y 539.088,Z 732.682,A -85,B 0,C 180,E1 25449.968,E2 25449.968} C_VEL
LIN {X 0,Y 539.608,Z 715.812,A -85,B 0,C 180,E1 25449.103,E2 25449.103} C_VEL
LIN {X 0,Y 540.086,Z 697.521,A -85,B 0,C 180,E1 25448.382,E2 25448.382} C_VEL
LIN {X 0,Y 540.462,Z 679.025,A -85,B 0,C 180,E1 25447.861,E2 25447.861} C_VEL
LIN {X 0,Y 540.681,Z 658.899,A -85,B 0,C 180,E1 25447.511,E2 25447.511} C_VEL
LIN {X 0,Y 541.413,Z 471.195,A -85,B 0,C 180,E1 25444.958,E2 25444.958} C_VEL
LIN {X 0,Y 540.147,Z 462.659,A -85,B 0,C 180,E1 25444.772,E2 25444.772} C_VEL
LIN {X 0,Y 541.28,Z 415.776,A -85,B 0,C 180,E1 25441.333,E2 25441.333} C_VEL
LIN {X 0,Y 542.282,Z 377.224,A -85,B 0,C 180,E1 25438.423,E2 25438.423} C_VEL
LIN {X 0,Y 536.389,Z 359.984,A -85,B 0,C 180,E1 25436.626,E2 25436.626} C_VEL
LIN {X 0,Y 536.418,Z 359.978,A -85,B 0,C 180,E1 25433.249,E2 25433.249} C_VEL
LIN {X 0,Y 536.407,Z 359.98,A -85,B 0,C 180,E1 25430.117,E2 25430.117} C_VEL
LIN {X 0,Y 536.391,Z 359.979,A -85,B 0,C 180,E1 25426.789,E2 25426.789} C_VEL
LIN {X 0,Y 536.454,Z 359.978,A -85,B 0,C 180,E1 25423.528,E2 25423.528} C_VEL
LIN {X 0,Y 536.388,Z 359.98,A -85,B 0,C 180,E1 25420.303,E2 25420.303} C_VEL
LIN {X 0,Y 536.4,Z 359.98,A -85,B 0,C 180,E1 25416.885,E2 25416.885} C_VEL
LIN {X 0,Y 536.421,Z 359.982,A -85,B 0,C 180,E1 25413.742,E2 25413.742} C_VEL
LIN {X 0,Y 536.383,Z 359.986,A -85,B 0,C 180,E1 25410.466,E2 25410.466} C_VEL
LIN {X 0,Y 536.464,Z 360.132,A -85,B 0,C 180,E1 25409.495,E2 25409.495} C_VEL
LIN {X 0,Y 540.52,Z 374.281,A -85,B 0,C 180,E1 25408.025,E2 25408.025} C_VEL
LIN {X 0,Y 540.19,Z 395.398,A -85,B 0,C 180,E1 25406.137,E2 25406.137} C_VEL
LIN {X 0,Y 540.101,Z 405.906,A -85,B 0,C 180,E1 25405.224,E2 25405.224} C_VEL
LIN {X 0,Y 541.76,Z 416.149,A -85,B 0,C 180,E1 25404.983,E2 25404.983} C_VEL
LIN {X 0,Y 540.458,Z 613.751,A -85,B 0,C 180,E1 25402.184,E2 25402.184} C_VEL
LIN {X 0,Y 540.122,Z 633.822,A -85,B 0,C 180,E1 25401.678,E2 25401.678} C_VEL
LIN {X 0,Y 539.692,Z 652.116,A -85,B 0,C 180,E1 25401.007,E2 25401.007} C_VEL
LIN {X 0,Y 539.2,Z 669.347,A -85,B 0,C 180,E1 25400.176,E2 25400.176} C_VEL
LIN {X 0,Y 538.595,Z 687.213,A -85,B 0,C 180,E1 25399.07,E2 25399.07} C_VEL
LIN {X 0,Y 538.026,Z 703.108,A -85,B 0,C 180,E1 25397.856,E2 25397.856} C_VEL
LIN {X 0,Y 537.499,Z 717.398,A -85,B 0,C 180,E1 25396.536,E2 25396.536} C_VEL
LIN {X 0,Y 537.021,Z 731.319,A -85,B 0,C 180,E1 25394.999,E2 25394.999} C_VEL
LIN {X 0,Y 536.636,Z 743.695,A -85,B 0,C 180,E1 25393.358,E2 25393.358} C_VEL
LIN {X 0,Y 536.336,Z 754.486,A -85,B 0,C 180,E1 25391.615,E2 25391.615} C_VEL
LIN {X 0,Y 536.133,Z 763.784,A -85,B 0,C 180,E1 25389.771,E2 25389.771} C_VEL
LIN {X 0,Y 536.008,Z 771.571,A -85,B 0,C 180,E1 25387.826,E2 25387.826} C_VEL
LIN {X 0,Y 535.948,Z 777.483,A -85,B 0,C 180,E1 25385.889,E2 25385.889} C_VEL
LIN {X 0,Y 535.916,Z 781.561,A -85,B 0,C 180,E1 25383.958,E2 25383.958} C_VEL
LIN {X 0,Y 535.909,Z 784.139,A -85,B 0,C 180,E1 25381.924,E2 25381.924} C_VEL
LIN {X 0,Y 535.914,Z 784.996,A -85,B 0,C 180,E1 25380,E2 25380} C_VEL
LIN {X 0,Y 535.906,Z 784.126,A -85,B 0,C 180,E1 25377.968,E2 25377.968} C_VEL
LIN {X 0,Y 535.917,Z 781.531,A -85,B 0,C 180,E1 25375.934,E2 25375.934} C_VEL
LIN {X 0,Y 535.941,Z 777.435,A -85,B 0,C 180,E1 25374.003,E2 25374.003} C_VEL
LIN {X 0,Y 536.003,Z 771.506,A -85,B 0,C 180,E1 25372.065,E2 25372.065} C_VEL
LIN {X 0,Y 536.132,Z 763.699,A -85,B 0,C 180,E1 25370.12,E2 25370.12} C_VEL
LIN {X 0,Y 536.34,Z 754.378,A -85,B 0,C 180,E1 25368.276,E2 25368.276} C_VEL
LIN {X 0,Y 536.643,Z 743.556,A -85,B 0,C 180,E1 25366.532,E2 25366.532} C_VEL
LIN {X 0,Y 537.027,Z 731.147,A -85,B 0,C 180,E1 25364.891,E2 25364.891} C_VEL
LIN {X 0,Y 537.513,Z 716.984,A -85,B 0,C 180,E1 25363.333,E2 25363.333} C_VEL
LIN {X 0,Y 538.058,Z 702.195,A -85,B 0,C 180,E1 25361.977,E2 25361.977} C_VEL
LIN {X 0,Y 538.607,Z 686.889,A -85,B 0,C 180,E1 25360.817,E2 25360.817} C_VEL
LIN {X 0,Y 539.215,Z 668.935,A -85,B 0,C 180,E1 25359.711,E2 25359.711} C_VEL
LIN {X 0,Y 539.757,Z 650.321,A -85,B 0,C 180,E1 25358.825,E2 25358.825} C_VEL
LIN {X 0,Y 540.176,Z 632.05,A -85,B 0,C 180,E1 25358.173,E2 25358.173} C_VEL
LIN {X 0,Y 540.508,Z 612.802,A -85,B 0,C 180,E1 25357.698,E2 25357.698} C_VEL
LIN {X 0,Y 540.767,Z 568.958,A -85,B 0,C 180,E1 25357.065,E2 25357.065} C_VEL
LIN {X 0,Y 539.88,Z 561.362,A -85,B 0,C 180,E1 25356.922,E2 25356.922} C_VEL
LIN {X 0,Y 534.191,Z 541.487,A -85,B 0,C 180,E1 25356.398,E2 25356.398} C_VEL
LIN {X 0,Y 533.541,Z 534.959,A -85,B 0,C 180,E1 25356.275,E2 25356.275} C_VEL
LIN {X 0,Y 534.34,Z 414.956,A -85,B 0,C 180,E1 25354.528,E2 25354.528} C_VEL
LIN {X 0,Y 532.441,Z 404.734,A -85,B 0,C 180,E1 25354.262,E2 25354.262} C_VEL
LIN {X 0,Y 533.123,Z 376.663,A -85,B 0,C 180,E1 25351.673,E2 25351.673} C_VEL
LIN {X 0,Y 528.459,Z 360.972,A -85,B 0,C 180,E1 25349.908,E2 25349.908} C_VEL
LIN {X 0,Y 528.506,Z 360.968,A -85,B 0,C 180,E1 25346.726,E2 25346.726} C_VEL
LIN {X 0,Y 528.452,Z 360.968,A -85,B 0,C 180,E1 25343.416,E2 25343.416} C_VEL
LIN {X 0,Y 528.473,Z 360.968,A -85,B 0,C 180,E1 25340.019,E2 25340.019} C_VEL
LIN {X 0,Y 528.476,Z 360.967,A -85,B 0,C 180,E1 25336.912,E2 25336.912} C_VEL
LIN {X 0,Y 528.451,Z 360.967,A -85,B 0,C 180,E1 25333.528,E2 25333.528} C_VEL
LIN {X 0,Y 528.518,Z 360.966,A -85,B 0,C 180,E1 25330.316,E2 25330.316} C_VEL
LIN {X 0,Y 528.46,Z 360.967,A -85,B 0,C 180,E1 25327.019,E2 25327.019} C_VEL
LIN {X 0,Y 528.454,Z 360.967,A -85,B 0,C 180,E1 25323.537,E2 25323.537} C_VEL
LIN {X 0,Y 528.519,Z 360.967,A -85,B 0,C 180,E1 25320.214,E2 25320.214} C_VEL
LIN {X 0,Y 528.46,Z 360.966,A -85,B 0,C 180,E1 25316.885,E2 25316.885} C_VEL
LIN {X 0,Y 528.452,Z 360.966,A -85,B 0,C 180,E1 25313.412,E2 25313.412} C_VEL
LIN {X 0,Y 528.515,Z 360.966,A -85,B 0,C 180,E1 25310.14,E2 25310.14} C_VEL
LIN {X 0,Y 528.457,Z 360.965,A -85,B 0,C 180,E1 25306.827,E2 25306.827} C_VEL
LIN {X 0,Y 528.453,Z 360.965,A -85,B 0,C 180,E1 25303.346,E2 25303.346} C_VEL
LIN {X 0,Y 528.514,Z 360.967,A -85,B 0,C 180,E1 25300.023,E2 25300.023} C_VEL
LIN {X 0,Y 528.457,Z 360.966,A -85,B 0,C 180,E1 25296.737,E2 25296.737} C_VEL
LIN {X 0,Y 528.453,Z 360.965,A -85,B 0,C 180,E1 25293.254,E2 25293.254} C_VEL
LIN {X 0,Y 528.519,Z 360.966,A -85,B 0,C 180,E1 25290,E2 25290} C_VEL
LIN {X 0,Y 528.454,Z 360.965,A -85,B 0,C 180,E1 25286.637,E2 25286.637} C_VEL
LIN {X 0,Y 528.452,Z 360.965,A -85,B 0,C 180,E1 25283.154,E2 25283.154} C_VEL
LIN {X 0,Y 528.513,Z 360.967,A -85,B 0,C 180,E1 25279.867,E2 25279.867} C_VEL
LIN {X 0,Y 528.453,Z 360.966,A -85,B 0,C 180,E1 25276.536,E2 25276.536} C_VEL
LIN {X 0,Y 528.454,Z 360.966,A -85,B 0,C 180,E1 25273.06,E2 25273.06} C_VEL
LIN {X 0,Y 528.515,Z 360.967,A -85,B 0,C 180,E1 25269.745,E2 25269.745} C_VEL
LIN {X 0,Y 528.448,Z 360.966,A -85,B 0,C 180,E1 25266.586,E2 25266.586} C_VEL
LIN {X 0,Y 528.473,Z 360.967,A -85,B 0,C 180,E1 25263.237,E2 25263.237} C_VEL
LIN {X 0,Y 528.474,Z 360.966,A -85,B 0,C 180,E1 25260.058,E2 25260.058} C_VEL
LIN {X 0,Y 528.446,Z 360.968,A -85,B 0,C 180,E1 25256.722,E2 25256.722} C_VEL
LIN {X 0,Y 528.503,Z 360.969,A -85,B 0,C 180,E1 25253.42,E2 25253.42} C_VEL
LIN {X 0,Y 528.454,Z 360.968,A -85,B 0,C 180,E1 25250.19,E2 25250.19} C_VEL
LIN {X 0,Y 528.451,Z 360.968,A -85,B 0,C 180,E1 25246.756,E2 25246.756} C_VEL
LIN {X 0,Y 528.512,Z 360.967,A -85,B 0,C 180,E1 25243.522,E2 25243.522} C_VEL
LIN {X 0,Y 528.447,Z 360.968,A -85,B 0,C 180,E1 25240.314,E2 25240.314} C_VEL
LIN {X 0,Y 528.474,Z 360.969,A -85,B 0,C 180,E1 25236.988,E2 25236.988} C_VEL
LIN {X 0,Y 528.47,Z 360.97,A -85,B 0,C 180,E1 25233.797,E2 25233.797} C_VEL
LIN {X 0,Y 528.447,Z 360.972,A -85,B 0,C 180,E1 25230.469,E2 25230.469} C_VEL
LIN {X 0,Y 528.52,Z 361.086,A -85,B 0,C 180,E1 25229.433,E2 25229.433} C_VEL
LIN {X 0,Y 531.942,Z 374.661,A -85,B 0,C 180,E1 25227.542,E2 25227.542} C_VEL
LIN {X 0,Y 531.114,Z 402.772,A -85,B 0,C 180,E1 25224.172,E2 25224.172} C_VEL
LIN {X 0,Y 530.395,Z 430.68,A -85,B 0,C 180,E1 25220.873,E2 25220.873} C_VEL
LIN {X 0,Y 529.65,Z 461.388,A -85,B 0,C 180,E1 25217.297,E2 25217.297} C_VEL
LIN {X 0,Y 529.279,Z 480.795,A -85,B 0,C 180,E1 25215.099,E2 25215.099} C_VEL
LIN {X 0,Y 530.42,Z 490.746,A -85,B 0,C 180,E1 25214.907,E2 25214.907} C_VEL
LIN {X 0,Y 529.825,Z 590.531,A -85,B 0,C 180,E1 25213.492,E2 25213.492} C_VEL
LIN {X 0,Y 529.691,Z 604.94,A -85,B 0,C 180,E1 25213.141,E2 25213.141} C_VEL
LIN {X 0,Y 529.479,Z 620.124,A -85,B 0,C 180,E1 25212.543,E2 25212.543} C_VEL
LIN {X 0,Y 529.205,Z 632.78,A -85,B 0,C 180,E1 25211.848,E2 25211.848} C_VEL
LIN {X 0,Y 528.899,Z 645.395,A -85,B 0,C 180,E1 25210.952,E2 25210.952} C_VEL
LIN {X 0,Y 528.657,Z 656.638,A -85,B 0,C 180,E1 25209.911,E2 25209.911} C_VEL
LIN {X 0,Y 528.431,Z 666.104,A -85,B 0,C 180,E1 25208.816,E2 25208.816} C_VEL
LIN {X 0,Y 528.239,Z 675.125,A -85,B 0,C 180,E1 25207.505,E2 25207.505} C_VEL
LIN {X 0,Y 528.115,Z 682.025,A -85,B 0,C 180,E1 25206.195,E2 25206.195} C_VEL
LIN {X 0,Y 528.032,Z 687.343,A -85,B 0,C 180,E1 25204.888,E2 25204.888} C_VEL
LIN {X 0,Y 527.982,Z 691.847,A -85,B 0,C 180,E1 25203.366,E2 25203.366} C_VEL
LIN {X 0,Y 527.961,Z 694.528,A -85,B 0,C 180,E1 25201.845,E2 25201.845} C_VEL
LIN {X 0,Y 527.961,Z 695.651,A -85,B 0,C 180,E1 25200.434,E2 25200.434} C_VEL
LIN {X 0,Y 527.961,Z 695.391,A -85,B 0,C 180,E1 25198.806,E2 25198.806} C_VEL
LIN {X 0,Y 527.982,Z 693.222,A -85,B 0,C 180,E1 25197.178,E2 25197.178} C_VEL
LIN {X 0,Y 528.021,Z 689.899,A -85,B 0,C 180,E1 25195.765,E2 25195.765} C_VEL
LIN {X 0,Y 528.121,Z 684.162,A -85,B 0,C 180,E1 25194.132,E2 25194.132} C_VEL
LIN {X 0,Y 528.233,Z 677.795,A -85,B 0,C 180,E1 25192.824,E2 25192.824} C_VEL
LIN {X 0,Y 528.414,Z 669.665,A -85,B 0,C 180,E1 25191.513,E2 25191.513} C_VEL
LIN {X 0,Y 528.666,Z 659.585,A -85,B 0,C 180,E1 25190.255,E2 25190.255} C_VEL
LIN {X 0,Y 528.928,Z 649.007,A -85,B 0,C 180,E1 25189.214,E2 25189.214} C_VEL
LIN {X 0,Y 529.211,Z 637.035,A -85,B 0,C 180,E1 25188.282,E2 25188.282} C_VEL
LIN {X 0,Y 529.514,Z 623.972,A -85,B 0,C 180,E1 25187.508,E2 25187.508} C_VEL
LIN {X 0,Y 529.754,Z 610.335,A -85,B 0,C 180,E1 25186.91,E2 25186.91} C_VEL
LIN {X 0,Y 529.946,Z 595.082,A -85,B 0,C 180,E1 25186.463,E2 25186.463} C_VEL
LIN {X 0,Y 530.723,Z 487.265,A -85,B 0,C 180,E1 25184.785,E2 25184.785} C_VEL
LIN {X 0,Y 529.55,Z 480.203,A -85,B 0,C 180,E1 25184.591,E2 25184.591} C_VEL
LIN {X 0,Y 530.364,Z 449.752,A -85,B 0,C 180,E1 25181.015,E2 25181.015} C_VEL
LIN {X 0,Y 531.276,Z 421.127,A -85,B 0,C 180,E1 25177.598,E2 25177.598} C_VEL
LIN {X 0,Y 532.379,Z 392.034,A -85,B 0,C 180,E1 25174.049,E2 25174.049} C_VEL
LIN {X 0,Y 532.949,Z 376.34,A -85,B 0,C 180,E1 25172.085,E2 25172.085} C_VEL
LIN {X 0,Y 529.171,Z 363.408,A -85,B 0,C 180,E1 25170.078,E2 25170.078} C_VEL
LIN {X 0,Y 528.447,Z 360.974,A -85,B 0,C 180,E1 25169.657,E2 25169.657} C_VEL
LIN {X 0,Y 528.491,Z 360.969,A -85,B 0,C 180,E1 25166.335,E2 25166.335} C_VEL
LIN {X 0,Y 528.46,Z 360.971,A -85,B 0,C 180,E1 25163.147,E2 25163.147} C_VEL
LIN {X 0,Y 528.455,Z 360.97,A -85,B 0,C 180,E1 25159.82,E2 25159.82} C_VEL
LIN {X 0,Y 528.509,Z 360.967,A -85,B 0,C 180,E1 25156.592,E2 25156.592} C_VEL
LIN {X 0,Y 528.449,Z 360.97,A -85,B 0,C 180,E1 25153.379,E2 25153.379} C_VEL
LIN {X 0,Y 528.481,Z 360.97,A -85,B 0,C 180,E1 25150.036,E2 25150.036} C_VEL
LIN {X 0,Y 528.473,Z 360.971,A -85,B 0,C 180,E1 25146.841,E2 25146.841} C_VEL
LIN {X 0,Y 528.494,Z 361.057,A -85,B 0,C 180,E1 25143.958,E2 25143.958} C_VEL
LIN {X 0,Y 533.957,Z 376.855,A -85,B 0,C 180,E1 25142.128,E2 25142.128} C_VEL
LIN {X 0,Y 534.922,Z 380.678,A -85,B 0,C 180,E1 25141.737,E2 25141.737} C_VEL
LIN {X 0,Y 533.65,Z 416.086,A -85,B 0,C 180,E1 25138.957,E2 25138.957} C_VEL
LIN {X 0,Y 532.508,Z 459.888,A -85,B 0,C 180,E1 25135.705,E2 25135.705} C_VEL
LIN {X 0,Y 532.504,Z 463.841,A -85,B 0,C 180,E1 25135.447,E2 25135.447} C_VEL
LIN {X 0,Y 533.911,Z 474.944,A -85,B 0,C 180,E1 25135.236,E2 25135.236} C_VEL
LIN {X 0,Y 532.875,Z 672.086,A -85,B 0,C 180,E1 25132.517,E2 25132.517} C_VEL
LIN {X 0,Y 532.539,Z 691.307,A -85,B 0,C 180,E1 25132.052,E2 25132.052} C_VEL
LIN {X 0,Y 532.104,Z 709.698,A -85,B 0,C 180,E1 25131.41,E2 25131.41} C_VEL
LIN {X 0,Y 531.605,Z 727.439,A -85,B 0,C 180,E1 25130.592,E2 25130.592} C_VEL
LIN {X 0,Y 531.112,Z 742.887,A -85,B 0,C 180,E1 25129.693,E2 25129.693} C_VEL
LIN {X 0,Y 530.511,Z 758.47,A -85,B 0,C 180,E1 25128.557,E2 25128.557} C_VEL
LIN {X 0,Y 529.897,Z 773.437,A -85,B 0,C 180,E1 25127.232,E2 25127.232} C_VEL
LIN {X 0,Y 529.35,Z 787.089,A -85,B 0,C 180,E1 25125.783,E2 25125.783} C_VEL
LIN {X 0,Y 528.892,Z 799.368,A -85,B 0,C 180,E1 25124.227,E2 25124.227} C_VEL
LIN {X 0,Y 528.504,Z 810.956,A -85,B 0,C 180,E1 25122.455,E2 25122.455} C_VEL
LIN {X 0,Y 528.245,Z 820.447,A -85,B 0,C 180,E1 25120.69,E2 25120.69} C_VEL
LIN {X 0,Y 528.066,Z 828.557,A -85,B 0,C 180,E1 25118.822,E2 25118.822} C_VEL
LIN {X 0,Y 527.971,Z 835.202,A -85,B 0,C 180,E1 25116.852,E2 25116.852} C_VEL
LIN {X 0,Y 527.931,Z 840.05,A -85,B 0,C 180,E1 25114.889,E2 25114.889} C_VEL
LIN {X 0,Y 527.913,Z 843.224,A -85,B 0,C 180,E1 25112.931,E2 25112.931} C_VEL
LIN {X 0,Y 527.916,Z 844.826,A -85,B 0,C 180,E1 25110.868,E2 25110.868} C_VEL
LIN {X 0,Y 527.914,Z 844.685,A -85,B 0,C 180,E1 25108.806,E2 25108.806} C_VEL
LIN {X 0,Y 527.913,Z 842.798,A -85,B 0,C 180,E1 25106.743,E2 25106.743} C_VEL
LIN {X 0,Y 527.935,Z 839.364,A -85,B 0,C 180,E1 25104.784,E2 25104.784} C_VEL
LIN {X 0,Y 527.988,Z 834.229,A -85,B 0,C 180,E1 25102.82,E2 25102.82} C_VEL
LIN {X 0,Y 528.097,Z 827.258,A -85,B 0,C 180,E1 25100.849,E2 25100.849} C_VEL
LIN {X 0,Y 528.283,Z 818.808,A -85,B 0,C 180,E1 25098.98,E2 25098.98} C_VEL
LIN {X 0,Y 528.568,Z 808.951,A -85,B 0,C 180,E1 25097.213,E2 25097.213} C_VEL
LIN {X 0,Y 528.949,Z 797.727,A -85,B 0,C 180,E1 25095.551,E2 25095.551} C_VEL
LIN {X 0,Y 529.44,Z 784.624,A -85,B 0,C 180,E1 25093.938,E2 25093.938} C_VEL
LIN {X 0,Y 530.006,Z 770.47,A -85,B 0,C 180,E1 25092.488,E2 25092.488} C_VEL
LIN {X 0,Y 530.625,Z 755.38,A -85,B 0,C 180,E1 25091.203,E2 25091.203} C_VEL
LIN {X 0,Y 531.211,Z 740.23,A -85,B 0,C 180,E1 25090.139,E2 25090.139} C_VEL
LIN {X 0,Y 531.722,Z 724.258,A -85,B 0,C 180,E1 25089.24,E2 25089.24} C_VEL
LIN {X 0,Y 532.216,Z 706.398,A -85,B 0,C 180,E1 25088.446,E2 25088.446} C_VEL
LIN {X 0,Y 532.643,Z 687.503,A -85,B 0,C 180,E1 25087.822,E2 25087.822} C_VEL
LIN {X 0,Y 532.967,Z 668.43,A -85,B 0,C 180,E1 25087.398,E2 25087.398} C_VEL
LIN {X 0,Y 533.938,Z 472.23,A -85,B 0,C 180,E1 25084.666,E2 25084.666} C_VEL
LIN {X 0,Y 532.562,Z 462.777,A -85,B 0,C 180,E1 25084.462,E2 25084.462} C_VEL
LIN {X 0,Y 533.84,Z 416.423,A -85,B 0,C 180,E1 25081.006,E2 25081.006} C_VEL
LIN {X 0,Y 534.982,Z 379.915,A -85,B 0,C 180,E1 25078.194,E2 25078.194} C_VEL
LIN {X 0,Y 528.468,Z 360.972,A -85,B 0,C 180,E1 25076.203,E2 25076.203} C_VEL
LIN {X 0,Y 528.451,Z 360.969,A -85,B 0,C 180,E1 25072.802,E2 25072.802} C_VEL
LIN {X 0,Y 528.516,Z 360.967,A -85,B 0,C 180,E1 25069.509,E2 25069.509} C_VEL
LIN {X 0,Y 528.459,Z 360.969,A -85,B 0,C 180,E1 25066.173,E2 25066.173} C_VEL
LIN {X 0,Y 528.452,Z 360.969,A -85,B 0,C 180,E1 25062.767,E2 25062.767} C_VEL
LIN {X 0,Y 528.524,Z 360.966,A -85,B 0,C 180,E1 25059.468,E2 25059.468} C_VEL
LIN {X 0,Y 528.454,Z 360.97,A -85,B 0,C 180,E1 25056.108,E2 25056.108} C_VEL
LIN {X 0,Y 528.45,Z 360.974,A -85,B 0,C 180,E1 25052.632,E2 25052.632} C_VEL
LIN {X 0,Y 528.483,Z 361.122,A -85,B 0,C 180,E1 25049.889,E2 25049.889} C_VEL
LIN {X 0,Y 533.104,Z 377.326,A -85,B 0,C 180,E1 25048.175,E2 25048.175} C_VEL
LIN {X 0,Y 532.739,Z 406.626,A -85,B 0,C 180,E1 25045.589,E2 25045.589} C_VEL
LIN {X 0,Y 534.505,Z 417.332,A -85,B 0,C 180,E1 25045.329,E2 25045.329} C_VEL
LIN {X 0,Y 533.145,Z 574.483,A -85,B 0,C 180,E1 25043.04,E2 25043.04} C_VEL
LIN {X 0,Y 532.868,Z 615.161,A -85,B 0,C 180,E1 25042.436,E2 25042.436} C_VEL
LIN {X 0,Y 532.529,Z 634.417,A -85,B 0,C 180,E1 25041.94,E2 25041.94} C_VEL
LIN {X 0,Y 532.077,Z 652.618,A -85,B 0,C 180,E1 25041.265,E2 25041.265} C_VEL
LIN {X 0,Y 531.544,Z 669.856,A -85,B 0,C 180,E1 25040.422,E2 25040.422} C_VEL
LIN {X 0,Y 530.933,Z 687.113,A -85,B 0,C 180,E1 25039.353,E2 25039.353} C_VEL
LIN {X 0,Y 530.311,Z 703.095,A -85,B 0,C 180,E1 25038.125,E2 25038.125} C_VEL
LIN {X 0,Y 529.718,Z 717.403,A -85,B 0,C 180,E1 25036.786,E2 25036.786} C_VEL
LIN {X 0,Y 529.175,Z 731.317,A -85,B 0,C 180,E1 25035.226,E2 25035.226} C_VEL
LIN {X 0,Y 528.749,Z 743.466,A -85,B 0,C 180,E1 25033.597,E2 25033.597} C_VEL
LIN {X 0,Y 528.401,Z 754.487,A -85,B 0,C 180,E1 25031.792,E2 25031.792} C_VEL
LIN {X 0,Y 528.179,Z 763.289,A -85,B 0,C 180,E1 25030.03,E2 25030.03} C_VEL
LIN {X 0,Y 528.032,Z 770.84,A -85,B 0,C 180,E1 25028.164,E2 25028.164} C_VEL
LIN {X 0,Y 527.954,Z 776.887,A -85,B 0,C 180,E1 25026.197,E2 25026.197} C_VEL
LIN {X 0,Y 527.915,Z 781.177,A -85,B 0,C 180,E1 25024.236,E2 25024.236} C_VEL
LIN {X 0,Y 527.911,Z 783.887,A -85,B 0,C 180,E1 25022.279,E2 25022.279} C_VEL
LIN {X 0,Y 527.908,Z 784.952,A -85,B 0,C 180,E1 25020.217,E2 25020.217} C_VEL
LIN {X 0,Y 527.906,Z 784.283,A -85,B 0,C 180,E1 25018.155,E2 25018.155} C_VEL
LIN {X 0,Y 527.915,Z 782.098,A -85,B 0,C 180,E1 25016.199,E2 25016.199} C_VEL
LIN {X 0,Y 527.937,Z 778.198,A -85,B 0,C 180,E1 25014.239,E2 25014.239} C_VEL
LIN {X 0,Y 528.006,Z 772.596,A -85,B 0,C 180,E1 25012.273,E2 25012.273} C_VEL
LIN {X 0,Y 528.126,Z 765.654,A -85,B 0,C 180,E1 25010.409,E2 25010.409} C_VEL
LIN {X 0,Y 528.339,Z 756.752,A -85,B 0,C 180,E1 25008.538,E2 25008.538} C_VEL
LIN {X 0,Y 528.64,Z 746.405,A -85,B 0,C 180,E1 25006.77,E2 25006.77} C_VEL
LIN {X 0,Y 529.052,Z 734.701,A -85,B 0,C 180,E1 25005.106,E2 25005.106} C_VEL
LIN {X 0,Y 529.567,Z 721.5,A -85,B 0,C 180,E1 25003.548,E2 25003.548} C_VEL
LIN {X 0,Y 530.172,Z 706.728,A -85,B 0,C 180,E1 25002.097,E2 25002.097} C_VEL
LIN {X 0,Y 530.807,Z 690.721,A -85,B 0,C 180,E1 25000.81,E2 25000.81} C_VEL
LIN {X 0,Y 531.404,Z 674.493,A -85,B 0,C 180,E1 24999.745,E2 24999.745} C_VEL
LIN {X 0,Y 532.003,Z 656.65,A -85,B 0,C 180,E1 24998.81,E2 24998.81} C_VEL
LIN {X 0,Y 532.506,Z 637.821,A -85,B 0,C 180,E1 24998.062,E2 24998.062} C_VEL
LIN {X 0,Y 532.906,Z 618.88,A -85,B 0,C 180,E1 24997.527,E2 24997.527} C_VEL
LIN {X 0,Y 533.147,Z 597.039,A -85,B 0,C 180,E1 24997.15,E2 24997.15} C_VEL
LIN {X 0,Y 533.541,Z 534.959,A -85,B 0,C 180,E1 24996.275,E2 24996.275} C_VEL
LIN {X 0,Y 532.681,Z 527.367,A -85,B 0,C 180,E1 24996.124,E2 24996.124} C_VEL
LIN {X 0,Y 527.091,Z 507.506,A -85,B 0,C 180,E1 24995.574,E2 24995.574} C_VEL
LIN {X 0,Y 526.473,Z 500.979,A -85,B 0,C 180,E1 24995.447,E2 24995.447} C_VEL
LIN {X 0,Y 527.099,Z 416.095,A -85,B 0,C 180,E1 24994.17,E2 24994.17} C_VEL
LIN {X 0,Y 525.042,Z 405.026,A -85,B 0,C 180,E1 24993.872,E2 24993.872} C_VEL
LIN {X 0,Y 525.695,Z 379.242,A -85,B 0,C 180,E1 24991.484,E2 24991.484} C_VEL
LIN {X 0,Y 520.514,Z 361.962,A -85,B 0,C 180,E1 24989.528,E2 24989.528} C_VEL
LIN {X 0,Y 520.54,Z 361.957,A -85,B 0,C 180,E1 24986.149,E2 24986.149} C_VEL
LIN {X 0,Y 520.549,Z 361.957,A -85,B 0,C 180,E1 24982.857,E2 24982.857} C_VEL
LIN {X 0,Y 520.514,Z 361.956,A -85,B 0,C 180,E1 24979.525,E2 24979.525} C_VEL
LIN {X 0,Y 520.561,Z 361.957,A -85,B 0,C 180,E1 24976.236,E2 24976.236} C_VEL
LIN {X 0,Y 520.529,Z 361.955,A -85,B 0,C 180,E1 24972.958,E2 24972.958} C_VEL
LIN {X 0,Y 520.516,Z 361.956,A -85,B 0,C 180,E1 24969.621,E2 24969.621} C_VEL
LIN {X 0,Y 520.576,Z 361.956,A -85,B 0,C 180,E1 24966.405,E2 24966.405} C_VEL
LIN {X 0,Y 520.517,Z 361.956,A -85,B 0,C 180,E1 24963.061,E2 24963.061} C_VEL
LIN {X 0,Y 520.515,Z 361.955,A -85,B 0,C 180,E1 24959.521,E2 24959.521} C_VEL
LIN {X 0,Y 520.576,Z 361.955,A -85,B 0,C 180,E1 24956.216,E2 24956.216} C_VEL
LIN {X 0,Y 520.516,Z 361.955,A -85,B 0,C 180,E1 24952.951,E2 24952.951} C_VEL
LIN {X 0,Y 520.515,Z 361.956,A -85,B 0,C 180,E1 24949.41,E2 24949.41} C_VEL
LIN {X 0,Y 520.574,Z 361.957,A -85,B 0,C 180,E1 24946.056,E2 24946.056} C_VEL
LIN {X 0,Y 520.513,Z 361.954,A -85,B 0,C 180,E1 24942.875,E2 24942.875} C_VEL
LIN {X 0,Y 520.519,Z 361.954,A -85,B 0,C 180,E1 24939.397,E2 24939.397} C_VEL
LIN {X 0,Y 520.578,Z 361.955,A -85,B 0,C 180,E1 24936.064,E2 24936.064} C_VEL
LIN {X 0,Y 520.515,Z 361.953,A -85,B 0,C 180,E1 24932.719,E2 24932.719} C_VEL
LIN {X 0,Y 520.515,Z 361.954,A -85,B 0,C 180,E1 24929.23,E2 24929.23} C_VEL
LIN {X 0,Y 520.573,Z 361.955,A -85,B 0,C 180,E1 24925.925,E2 24925.925} C_VEL
LIN {X 0,Y 520.514,Z 361.954,A -85,B 0,C 180,E1 24922.605,E2 24922.605} C_VEL
LIN {X 0,Y 520.516,Z 361.956,A -85,B 0,C 180,E1 24919.149,E2 24919.149} C_VEL
LIN {X 0,Y 520.582,Z 361.956,A -85,B 0,C 180,E1 24915.768,E2 24915.768} C_VEL
LIN {X 0,Y 520.517,Z 361.955,A -85,B 0,C 180,E1 24912.447,E2 24912.447} C_VEL
LIN {X 0,Y 520.512,Z 361.955,A -85,B 0,C 180,E1 24908.948,E2 24908.948} C_VEL
LIN {X 0,Y 520.573,Z 361.955,A -85,B 0,C 180,E1 24905.73,E2 24905.73} C_VEL
LIN {X 0,Y 520.513,Z 361.955,A -85,B 0,C 180,E1 24902.423,E2 24902.423} C_VEL
LIN {X 0,Y 520.513,Z 361.957,A -85,B 0,C 180,E1 24898.887,E2 24898.887} C_VEL
LIN {X 0,Y 520.57,Z 361.958,A -85,B 0,C 180,E1 24895.619,E2 24895.619} C_VEL
LIN {X 0,Y 520.511,Z 361.958,A -85,B 0,C 180,E1 24892.319,E2 24892.319} C_VEL
LIN {X 0,Y 520.512,Z 361.956,A -85,B 0,C 180,E1 24888.786,E2 24888.786} C_VEL
LIN {X 0,Y 520.573,Z 361.956,A -85,B 0,C 180,E1 24885.445,E2 24885.445} C_VEL
LIN {X 0,Y 520.517,Z 361.957,A -85,B 0,C 180,E1 24882.098,E2 24882.098} C_VEL
LIN {X 0,Y 520.51,Z 361.958,A -85,B 0,C 180,E1 24878.631,E2 24878.631} C_VEL
LIN {X 0,Y 520.567,Z 361.958,A -85,B 0,C 180,E1 24875.283,E2 24875.283} C_VEL
LIN {X 0,Y 520.515,Z 361.96,A -85,B 0,C 180,E1 24872.017,E2 24872.017} C_VEL
LIN {X 0,Y 520.541,Z 362.075,A -85,B 0,C 180,E1 24869.803,E2 24869.803} C_VEL
LIN {X 0,Y 524.378,Z 377.19,A -85,B 0,C 180,E1 24867.665,E2 24867.665} C_VEL
LIN {X 0,Y 523.449,Z 405.349,A -85,B 0,C 180,E1 24864.248,E2 24864.248} C_VEL
LIN {X 0,Y 522.637,Z 433.792,A -85,B 0,C 180,E1 24860.845,E2 24860.845} C_VEL
LIN {X 0,Y 521.817,Z 464.468,A -85,B 0,C 180,E1 24857.235,E2 24857.235} C_VEL
LIN {X 0,Y 521.49,Z 480.666,A -85,B 0,C 180,E1 24855.379,E2 24855.379} C_VEL
LIN {X 0,Y 522.796,Z 491.477,A -85,B 0,C 180,E1 24855.163,E2 24855.163} C_VEL
LIN {X 0,Y 522.067,Z 593.531,A -85,B 0,C 180,E1 24853.661,E2 24853.661} C_VEL
LIN {X 0,Y 521.898,Z 608.866,A -85,B 0,C 180,E1 24853.235,E2 24853.235} C_VEL
LIN {X 0,Y 521.66,Z 623.126,A -85,B 0,C 180,E1 24852.621,E2 24852.621} C_VEL
LIN {X 0,Y 521.34,Z 636.479,A -85,B 0,C 180,E1 24851.842,E2 24851.842} C_VEL
LIN {X 0,Y 521.024,Z 648.776,A -85,B 0,C 180,E1 24850.896,E2 24850.896} C_VEL
LIN {X 0,Y 520.764,Z 659.566,A -85,B 0,C 180,E1 24849.839,E2 24849.839} C_VEL
LIN {X 0,Y 520.513,Z 669.523,A -85,B 0,C 180,E1 24848.617,E2 24848.617} C_VEL
LIN {X 0,Y 520.321,Z 677.958,A -85,B 0,C 180,E1 24847.286,E2 24847.286} C_VEL
LIN {X 0,Y 520.185,Z 685.021,A -85,B 0,C 180,E1 24845.847,E2 24845.847} C_VEL
LIN {X 0,Y 520.097,Z 690.574,A -85,B 0,C 180,E1 24844.3,E2 24844.3} C_VEL
LIN {X 0,Y 520.059,Z 694.271,A -85,B 0,C 180,E1 24842.755,E2 24842.755} C_VEL
LIN {X 0,Y 520.044,Z 696.441,A -85,B 0,C 180,E1 24841.2,E2 24841.2} C_VEL
LIN {X 0,Y 520.053,Z 696.881,A -85,B 0,C 180,E1 24839.449,E2 24839.449} C_VEL
LIN {X 0,Y 520.069,Z 695.679,A -85,B 0,C 180,E1 24837.907,E2 24837.907} C_VEL
LIN {X 0,Y 520.116,Z 692.61,A -85,B 0,C 180,E1 24836.253,E2 24836.253} C_VEL
LIN {X 0,Y 520.198,Z 687.921,A -85,B 0,C 180,E1 24834.707,E2 24834.707} C_VEL
LIN {X 0,Y 520.322,Z 681.904,A -85,B 0,C 180,E1 24833.269,E2 24833.269} C_VEL
LIN {X 0,Y 520.517,Z 673.801,A -85,B 0,C 180,E1 24831.828,E2 24831.828} C_VEL
LIN {X 0,Y 520.751,Z 665.013,A -85,B 0,C 180,E1 24830.607,E2 24830.607} C_VEL
LIN {X 0,Y 521.064,Z 653.811,A -85,B 0,C 180,E1 24829.385,E2 24829.385} C_VEL
LIN {X 0,Y 521.378,Z 641.301,A -85,B 0,C 180,E1 24828.327,E2 24828.327} C_VEL
LIN {X 0,Y 521.711,Z 628.406,A -85,B 0,C 180,E1 24827.493,E2 24827.493} C_VEL
LIN {X 0,Y 521.993,Z 614.586,A -85,B 0,C 180,E1 24826.824,E2 24826.824} C_VEL
LIN {X 0,Y 522.224,Z 599.072,A -85,B 0,C 180,E1 24826.311,E2 24826.311} C_VEL
LIN {X 0,Y 522.396,Z 577.868,A -85,B 0,C 180,E1 24825.928,E2 24825.928} C_VEL
LIN {X 0,Y 523.281,Z 488.12,A -85,B 0,C 180,E1 24824.474,E2 24824.474} C_VEL
LIN {X 0,Y 521.871,Z 480.345,A -85,B 0,C 180,E1 24824.27,E2 24824.27} C_VEL
LIN {X 0,Y 522.773,Z 450.16,A -85,B 0,C 180,E1 24820.678,E2 24820.678} C_VEL
LIN {X 0,Y 523.851,Z 420.838,A -85,B 0,C 180,E1 24817.121,E2 24817.121} C_VEL
LIN {X 0,Y 525.056,Z 393.008,A -85,B 0,C 180,E1 24813.66,E2 24813.66} C_VEL
LIN {X 0,Y 525.716,Z 379.516,A -85,B 0,C 180,E1 24811.944,E2 24811.944} C_VEL
LIN {X 0,Y 521.908,Z 366.564,A -85,B 0,C 180,E1 24809.872,E2 24809.872} C_VEL
LIN {X 0,Y 520.532,Z 361.961,A -85,B 0,C 180,E1 24809.081,E2 24809.081} C_VEL
LIN {X 0,Y 520.511,Z 361.961,A -85,B 0,C 180,E1 24805.69,E2 24805.69} C_VEL
LIN {X 0,Y 520.56,Z 361.958,A -85,B 0,C 180,E1 24802.353,E2 24802.353} C_VEL
LIN {X 0,Y 520.518,Z 361.959,A -85,B 0,C 180,E1 24799.186,E2 24799.186} C_VEL
LIN {X 0,Y 520.516,Z 361.96,A -85,B 0,C 180,E1 24795.766,E2 24795.766} C_VEL
LIN {X 0,Y 520.574,Z 361.956,A -85,B 0,C 180,E1 24792.478,E2 24792.478} C_VEL
LIN {X 0,Y 520.514,Z 361.96,A -85,B 0,C 180,E1 24789.197,E2 24789.197} C_VEL
LIN {X 0,Y 520.521,Z 361.961,A -85,B 0,C 180,E1 24785.729,E2 24785.729} C_VEL
LIN {X 0,Y 520.567,Z 362.029,A -85,B 0,C 180,E1 24784.552,E2 24784.552} C_VEL
LIN {X 0,Y 526.4,Z 378.598,A -85,B 0,C 180,E1 24782.505,E2 24782.505} C_VEL
LIN {X 0,Y 527.699,Z 383.563,A -85,B 0,C 180,E1 24781.978,E2 24781.978} C_VEL
LIN {X 0,Y 526.129,Z 419.843,A -85,B 0,C 180,E1 24779.051,E2 24779.051} C_VEL
LIN {X 0,Y 524.832,Z 462.994,A -85,B 0,C 180,E1 24775.789,E2 24775.789} C_VEL
LIN {X 0,Y 526.36,Z 475.898,A -85,B 0,C 180,E1 24775.511,E2 24775.511} C_VEL
LIN {X 0,Y 525.169,Z 671.503,A -85,B 0,C 180,E1 24772.758,E2 24772.758} C_VEL
LIN {X 0,Y 524.8,Z 690.562,A -85,B 0,C 180,E1 24772.292,E2 24772.292} C_VEL
LIN {X 0,Y 524.344,Z 708.318,A -85,B 0,C 180,E1 24771.668,E2 24771.668} C_VEL
LIN {X 0,Y 523.82,Z 725.879,A -85,B 0,C 180,E1 24770.854,E2 24770.854} C_VEL
LIN {X 0,Y 523.262,Z 742.533,A -85,B 0,C 180,E1 24769.885,E2 24769.885} C_VEL
LIN {X 0,Y 522.639,Z 759.215,A -85,B 0,C 180,E1 24768.69,E2 24768.69} C_VEL
LIN {X 0,Y 522.049,Z 774.638,A -85,B 0,C 180,E1 24767.348,E2 24767.348} C_VEL
LIN {X 0,Y 521.538,Z 787.089,A -85,B 0,C 180,E1 24766.026,E2 24766.026} C_VEL
LIN {X 0,Y 521.024,Z 799.369,A -85,B 0,C 180,E1 24764.446,E2 24764.446} C_VEL
LIN {X 0,Y 520.589,Z 810.956,A -85,B 0,C 180,E1 24762.648,E2 24762.648} C_VEL
LIN {X 0,Y 520.291,Z 820.448,A -85,B 0,C 180,E1 24760.855,E2 24760.855} C_VEL
LIN {X 0,Y 520.09,Z 828.557,A -85,B 0,C 180,E1 24758.959,E2 24758.959} C_VEL
LIN {X 0,Y 519.982,Z 835.202,A -85,B 0,C 180,E1 24756.958,E2 24756.958} C_VEL
LIN {X 0,Y 519.933,Z 840.05,A -85,B 0,C 180,E1 24754.964,E2 24754.964} C_VEL
LIN {X 0,Y 519.913,Z 843.223,A -85,B 0,C 180,E1 24752.976,E2 24752.976} C_VEL
LIN {X 0,Y 519.916,Z 844.825,A -85,B 0,C 180,E1 24750.882,E2 24750.882} C_VEL
LIN {X 0,Y 519.914,Z 844.685,A -85,B 0,C 180,E1 24748.788,E2 24748.788} C_VEL
LIN {X 0,Y 519.913,Z 842.798,A -85,B 0,C 180,E1 24746.693,E2 24746.693} C_VEL
LIN {X 0,Y 519.938,Z 839.365,A -85,B 0,C 180,E1 24744.704,E2 24744.704} C_VEL
LIN {X 0,Y 519.999,Z 834.228,A -85,B 0,C 180,E1 24742.709,E2 24742.709} C_VEL
LIN {X 0,Y 520.128,Z 827.257,A -85,B 0,C 180,E1 24740.707,E2 24740.707} C_VEL
LIN {X 0,Y 520.336,Z 818.807,A -85,B 0,C 180,E1 24738.809,E2 24738.809} C_VEL
LIN {X 0,Y 520.656,Z 808.949,A -85,B 0,C 180,E1 24737.016,E2 24737.016} C_VEL
LIN {X 0,Y 521.103,Z 797.135,A -85,B 0,C 180,E1 24735.249,E2 24735.249} C_VEL
LIN {X 0,Y 521.658,Z 784.102,A -85,B 0,C 180,E1 24733.635,E2 24733.635} C_VEL
LIN {X 0,Y 522.176,Z 771.269,A -85,B 0,C 180,E1 24732.332,E2 24732.332} C_VEL
LIN {X 0,Y 522.79,Z 755.743,A -85,B 0,C 180,E1 24731.026,E2 24731.026} C_VEL
LIN {X 0,Y 523.414,Z 739.341,A -85,B 0,C 180,E1 24729.888,E2 24729.888} C_VEL
LIN {X 0,Y 524.013,Z 722.021,A -85,B 0,C 180,E1 24728.915,E2 24728.915} C_VEL
LIN {X 0,Y 524.563,Z 703.968,A -85,B 0,C 180,E1 24728.121,E2 24728.121} C_VEL
LIN {X 0,Y 525.021,Z 685.082,A -85,B 0,C 180,E1 24727.508,E2 24727.508} C_VEL
LIN {X 0,Y 525.365,Z 665.177,A -85,B 0,C 180,E1 24727.084,E2 24727.084} C_VEL
LIN {X 0,Y 526.519,Z 473.506,A -85,B 0,C 180,E1 24724.37,E2 24724.37} C_VEL
LIN {X 0,Y 524.993,Z 462.892,A -85,B 0,C 180,E1 24724.142,E2 24724.142} C_VEL
LIN {X 0,Y 526.427,Z 417.766,A -85,B 0,C 180,E1 24720.714,E2 24720.714} C_VEL
LIN {X 0,Y 527.656,Z 382.603,A -85,B 0,C 180,E1 24717.956,E2 24717.956} C_VEL
LIN {X 0,Y 520.577,Z 361.956,A -85,B 0,C 180,E1 24715.716,E2 24715.716} C_VEL
LIN {X 0,Y 520.516,Z 361.959,A -85,B 0,C 180,E1 24712.349,E2 24712.349} C_VEL
LIN {X 0,Y 520.516,Z 361.958,A -85,B 0,C 180,E1 24708.85,E2 24708.85} C_VEL
LIN {X 0,Y 520.573,Z 361.957,A -85,B 0,C 180,E1 24705.488,E2 24705.488} C_VEL
LIN {X 0,Y 520.518,Z 361.959,A -85,B 0,C 180,E1 24702.143,E2 24702.143} C_VEL
LIN {X 0,Y 520.514,Z 361.959,A -85,B 0,C 180,E1 24698.749,E2 24698.749} C_VEL
LIN {X 0,Y 520.571,Z 361.957,A -85,B 0,C 180,E1 24695.454,E2 24695.454} C_VEL
LIN {X 0,Y 520.513,Z 361.963,A -85,B 0,C 180,E1 24692.147,E2 24692.147} C_VEL
LIN {X 0,Y 520.524,Z 362.104,A -85,B 0,C 180,E1 24690.321,E2 24690.321} C_VEL
LIN {X 0,Y 525.776,Z 379.302,A -85,B 0,C 180,E1 24688.449,E2 24688.449} C_VEL
LIN {X 0,Y 525.419,Z 407.495,A -85,B 0,C 180,E1 24685.958,E2 24685.958} C_VEL
LIN {X 0,Y 527.236,Z 418.569,A -85,B 0,C 180,E1 24685.677,E2 24685.677} C_VEL
LIN {X 0,Y 525.661,Z 568.353,A -85,B 0,C 180,E1 24683.424,E2 24683.424} C_VEL
LIN {X 0,Y 525.302,Z 615.488,A -85,B 0,C 180,E1 24682.715,E2 24682.715} C_VEL
LIN {X 0,Y 524.953,Z 634.604,A -85,B 0,C 180,E1 24682.22,E2 24682.22} C_VEL
LIN {X 0,Y 524.465,Z 653.037,A -85,B 0,C 180,E1 24681.53,E2 24681.53} C_VEL
LIN {X 0,Y 523.895,Z 670.322,A -85,B 0,C 180,E1 24680.675,E2 24680.675} C_VEL
LIN {X 0,Y 523.27,Z 686.76,A -85,B 0,C 180,E1 24679.651,E2 24679.651} C_VEL
LIN {X 0,Y 522.627,Z 702.323,A -85,B 0,C 180,E1 24678.459,E2 24678.459} C_VEL
LIN {X 0,Y 521.978,Z 717.009,A -85,B 0,C 180,E1 24677.089,E2 24677.089} C_VEL
LIN {X 0,Y 521.391,Z 730.522,A -85,B 0,C 180,E1 24675.573,E2 24675.573} C_VEL
LIN {X 0,Y 520.882,Z 742.973,A -85,B 0,C 180,E1 24673.883,E2 24673.883} C_VEL
LIN {X 0,Y 520.49,Z 753.854,A -85,B 0,C 180,E1 24672.086,E2 24672.086} C_VEL
LIN {X 0,Y 520.213,Z 763.286,A -85,B 0,C 180,E1 24670.185,E2 24670.185} C_VEL
LIN {X 0,Y 520.051,Z 770.838,A -85,B 0,C 180,E1 24668.291,E2 24668.291} C_VEL
LIN {X 0,Y 519.958,Z 776.887,A -85,B 0,C 180,E1 24666.293,E2 24666.293} C_VEL
LIN {X 0,Y 519.917,Z 781.174,A -85,B 0,C 180,E1 24664.301,E2 24664.301} C_VEL
LIN {X 0,Y 519.911,Z 783.887,A -85,B 0,C 180,E1 24662.314,E2 24662.314} C_VEL
LIN {X 0,Y 519.907,Z 784.922,A -85,B 0,C 180,E1 24660.33,E2 24660.33} C_VEL
LIN {X 0,Y 519.907,Z 784.359,A -85,B 0,C 180,E1 24658.237,E2 24658.237} C_VEL
LIN {X 0,Y 519.915,Z 782.265,A -85,B 0,C 180,E1 24656.251,E2 24656.251} C_VEL
LIN {X 0,Y 519.94,Z 778.441,A -85,B 0,C 180,E1 24654.261,E2 24654.261} C_VEL
LIN {X 0,Y 520.018,Z 772.589,A -85,B 0,C 180,E1 24652.154,E2 24652.154} C_VEL
LIN {X 0,Y 520.155,Z 765.652,A -85,B 0,C 180,E1 24650.261,E2 24650.261} C_VEL
LIN {X 0,Y 520.397,Z 756.744,A -85,B 0,C 180,E1 24648.361,E2 24648.361} C_VEL
LIN {X 0,Y 520.743,Z 746.396,A -85,B 0,C 180,E1 24646.566,E2 24646.566} C_VEL
LIN {X 0,Y 521.213,Z 734.738,A -85,B 0,C 180,E1 24644.877,E2 24644.877} C_VEL
LIN {X 0,Y 521.79,Z 721.544,A -85,B 0,C 180,E1 24643.296,E2 24643.296} C_VEL
LIN {X 0,Y 522.454,Z 706.664,A -85,B 0,C 180,E1 24641.823,E2 24641.823} C_VEL
LIN {X 0,Y 523.151,Z 690.565,A -85,B 0,C 180,E1 24640.518,E2 24640.518} C_VEL
LIN {X 0,Y 523.803,Z 674.171,A -85,B 0,C 180,E1 24639.437,E2 24639.437} C_VEL
LIN {X 0,Y 524.425,Z 656.907,A -85,B 0,C 180,E1 24638.527,E2 24638.527} C_VEL
LIN {X 0,Y 524.97,Z 638.177,A -85,B 0,C 180,E1 24637.772,E2 24637.772} C_VEL
LIN {X 0,Y 525.403,Z 619.048,A -85,B 0,C 180,E1 24637.225,E2 24637.225} C_VEL
LIN {X 0,Y 525.669,Z 597.714,A -85,B 0,C 180,E1 24636.848,E2 24636.848} C_VEL
LIN {X 0,Y 526.473,Z 500.979,A -85,B 0,C 180,E1 24635.447,E2 24635.447} C_VEL
LIN {X 0,Y 525.647,Z 493.391,A -85,B 0,C 180,E1 24635.293,E2 24635.293} C_VEL
LIN {X 0,Y 520.119,Z 473.562,A -85,B 0,C 180,E1 24634.713,E2 24634.713} C_VEL
LIN {X 0,Y 519.493,Z 467.04,A -85,B 0,C 180,E1 24634.58,E2 24634.58} C_VEL
LIN {X 0,Y 519.895,Z 417.386,A -85,B 0,C 180,E1 24633.805,E2 24633.805} C_VEL
LIN {X 0,Y 517.667,Z 405.285,A -85,B 0,C 180,E1 24633.468,E2 24633.468} C_VEL
LIN {X 0,Y 518.292,Z 381.92,A -85,B 0,C 180,E1 24631.291,E2 24631.291} C_VEL
LIN {X 0,Y 512.594,Z 362.95,A -85,B 0,C 180,E1 24629.122,E2 24629.122} C_VEL
LIN {X 0,Y 512.575,Z 362.947,A -85,B 0,C 180,E1 24625.685,E2 24625.685} C_VEL
LIN {X 0,Y 512.628,Z 362.943,A -85,B 0,C 180,E1 24622.363,E2 24622.363} C_VEL
LIN {X 0,Y 512.581,Z 362.945,A -85,B 0,C 180,E1 24619.187,E2 24619.187} C_VEL
LIN {X 0,Y 512.579,Z 362.946,A -85,B 0,C 180,E1 24615.707,E2 24615.707} C_VEL
LIN {X 0,Y 512.634,Z 362.946,A -85,B 0,C 180,E1 24612.335,E2 24612.335} C_VEL
LIN {X 0,Y 512.582,Z 362.944,A -85,B 0,C 180,E1 24609.054,E2 24609.054} C_VEL
LIN {X 0,Y 512.576,Z 362.946,A -85,B 0,C 180,E1 24605.542,E2 24605.542} C_VEL
LIN {X 0,Y 512.629,Z 362.945,A -85,B 0,C 180,E1 24602.167,E2 24602.167} C_VEL
LIN {X 0,Y 512.585,Z 362.944,A -85,B 0,C 180,E1 24598.856,E2 24598.856} C_VEL
LIN {X 0,Y 512.575,Z 362.945,A -85,B 0,C 180,E1 24595.413,E2 24595.413} C_VEL
LIN {X 0,Y 512.638,Z 362.944,A -85,B 0,C 180,E1 24592.111,E2 24592.111} C_VEL
LIN {X 0,Y 512.584,Z 362.944,A -85,B 0,C 180,E1 24588.775,E2 24588.775} C_VEL
LIN {X 0,Y 512.572,Z 362.945,A -85,B 0,C 180,E1 24585.268,E2 24585.268} C_VEL
LIN {X 0,Y 512.633,Z 362.945,A -85,B 0,C 180,E1 24582.046,E2 24582.046} C_VEL
LIN {X 0,Y 512.579,Z 362.942,A -85,B 0,C 180,E1 24578.752,E2 24578.752} C_VEL
LIN {X 0,Y 512.576,Z 362.944,A -85,B 0,C 180,E1 24575.26,E2 24575.26} C_VEL
LIN {X 0,Y 512.631,Z 362.946,A -85,B 0,C 180,E1 24571.9,E2 24571.9} C_VEL
LIN {X 0,Y 512.576,Z 362.942,A -85,B 0,C 180,E1 24568.659,E2 24568.659} C_VEL
LIN {X 0,Y 512.576,Z 362.945,A -85,B 0,C 180,E1 24565.188,E2 24565.188} C_VEL
LIN {X 0,Y 512.638,Z 362.942,A -85,B 0,C 180,E1 24561.927,E2 24561.927} C_VEL
LIN {X 0,Y 512.578,Z 362.944,A -85,B 0,C 180,E1 24558.523,E2 24558.523} C_VEL
LIN {X 0,Y 512.576,Z 362.945,A -85,B 0,C 180,E1 24555.079,E2 24555.079} C_VEL
LIN {X 0,Y 512.632,Z 362.947,A -85,B 0,C 180,E1 24551.698,E2 24551.698} C_VEL
LIN {X 0,Y 512.58,Z 362.944,A -85,B 0,C 180,E1 24548.366,E2 24548.366} C_VEL
LIN {X 0,Y 512.571,Z 362.945,A -85,B 0,C 180,E1 24544.839,E2 24544.839} C_VEL
LIN {X 0,Y 512.621,Z 362.945,A -85,B 0,C 180,E1 24541.453,E2 24541.453} C_VEL
LIN {X 0,Y 512.582,Z 362.945,A -85,B 0,C 180,E1 24538.219,E2 24538.219} C_VEL
LIN {X 0,Y 512.57,Z 362.947,A -85,B 0,C 180,E1 24534.732,E2 24534.732} C_VEL
LIN {X 0,Y 512.623,Z 362.947,A -85,B 0,C 180,E1 24531.38,E2 24531.38} C_VEL
LIN {X 0,Y 512.58,Z 362.944,A -85,B 0,C 180,E1 24528.155,E2 24528.155} C_VEL
LIN {X 0,Y 512.575,Z 362.946,A -85,B 0,C 180,E1 24524.761,E2 24524.761} C_VEL
LIN {X 0,Y 512.635,Z 362.946,A -85,B 0,C 180,E1 24521.391,E2 24521.391} C_VEL
LIN {X 0,Y 512.577,Z 362.947,A -85,B 0,C 180,E1 24518.054,E2 24518.054} C_VEL
LIN {X 0,Y 512.572,Z 362.948,A -85,B 0,C 180,E1 24514.586,E2 24514.586} C_VEL
LIN {X 0,Y 512.634,Z 362.945,A -85,B 0,C 180,E1 24511.253,E2 24511.253} C_VEL
LIN {X 0,Y 512.584,Z 363.055,A -85,B 0,C 180,E1 24510.184,E2 24510.184} C_VEL
LIN {X 0,Y 516.815,Z 379.711,A -85,B 0,C 180,E1 24507.792,E2 24507.792} C_VEL
LIN {X 0,Y 515.788,Z 407.799,A -85,B 0,C 180,E1 24504.342,E2 24504.342} C_VEL
LIN {X 0,Y 514.9,Z 435.995,A -85,B 0,C 180,E1 24500.927,E2 24500.927} C_VEL
LIN {X 0,Y 514.01,Z 466.295,A -85,B 0,C 180,E1 24497.315,E2 24497.315} C_VEL
LIN {X 0,Y 513.702,Z 480.462,A -85,B 0,C 180,E1 24495.669,E2 24495.669} C_VEL
LIN {X 0,Y 515.184,Z 492.241,A -85,B 0,C 180,E1 24495.427,E2 24495.427} C_VEL
LIN {X 0,Y 514.32,Z 595.149,A -85,B 0,C 180,E1 24493.855,E2 24493.855} C_VEL
LIN {X 0,Y 514.133,Z 610.381,A -85,B 0,C 180,E1 24493.41,E2 24493.41} C_VEL
LIN {X 0,Y 513.868,Z 625.014,A -85,B 0,C 180,E1 24492.759,E2 24492.759} C_VEL
LIN {X 0,Y 513.502,Z 638.86,A -85,B 0,C 180,E1 24491.911,E2 24491.911} C_VEL
LIN {X 0,Y 513.176,Z 650.832,A -85,B 0,C 180,E1 24490.951,E2 24490.951} C_VEL
LIN {X 0,Y 512.874,Z 662.464,A -85,B 0,C 180,E1 24489.765,E2 24489.765} C_VEL
LIN {X 0,Y 512.593,Z 672.752,A -85,B 0,C 180,E1 24488.412,E2 24488.412} C_VEL
LIN {X 0,Y 512.399,Z 680.746,A -85,B 0,C 180,E1 24487.062,E2 24487.062} C_VEL
LIN {X 0,Y 512.254,Z 687.846,A -85,B 0,C 180,E1 24485.488,E2 24485.488} C_VEL
LIN {X 0,Y 512.171,Z 692.871,A -85,B 0,C 180,E1 24483.918,E2 24483.918} C_VEL
LIN {X 0,Y 512.134,Z 696.215,A -85,B 0,C 180,E1 24482.35,E2 24482.35} C_VEL
LIN {X 0,Y 512.139,Z 697.95,A -85,B 0,C 180,E1 24480.671,E2 24480.671} C_VEL
LIN {X 0,Y 512.144,Z 697.904,A -85,B 0,C 180,E1 24478.993,E2 24478.993} C_VEL
LIN {X 0,Y 512.182,Z 696.078,A -85,B 0,C 180,E1 24477.315,E2 24477.315} C_VEL
LIN {X 0,Y 512.255,Z 692.373,A -85,B 0,C 180,E1 24475.634,E2 24475.634} C_VEL
LIN {X 0,Y 512.39,Z 686.595,A -85,B 0,C 180,E1 24473.951,E2 24473.951} C_VEL
LIN {X 0,Y 512.56,Z 679.621,A -85,B 0,C 180,E1 24472.49,E2 24472.49} C_VEL
LIN {X 0,Y 512.792,Z 671.268,A -85,B 0,C 180,E1 24471.139,E2 24471.139} C_VEL
LIN {X 0,Y 513.106,Z 660.92,A -85,B 0,C 180,E1 24469.843,E2 24469.843} C_VEL
LIN {X 0,Y 513.418,Z 650.082,A -85,B 0,C 180,E1 24468.77,E2 24468.77} C_VEL
LIN {X 0,Y 513.784,Z 636.906,A -85,B 0,C 180,E1 24467.753,E2 24467.753} C_VEL
LIN {X 0,Y 514.157,Z 622.162,A -85,B 0,C 180,E1 24466.906,E2 24466.906} C_VEL
LIN {X 0,Y 514.425,Z 606.963,A -85,B 0,C 180,E1 24466.291,E2 24466.291} C_VEL
LIN {X 0,Y 514.603,Z 592.072,A -85,B 0,C 180,E1 24465.908,E2 24465.908} C_VEL
LIN {X 0,Y 515.846,Z 489.016,A -85,B 0,C 180,E1 24464.155,E2 24464.155} C_VEL
LIN {X 0,Y 514.21,Z 480.298,A -85,B 0,C 180,E1 24463.914,E2 24463.914} C_VEL
LIN {X 0,Y 515.247,Z 449.984,A -85,B 0,C 180,E1 24460.249,E2 24460.249} C_VEL
LIN {X 0,Y 516.51,Z 420.233,A -85,B 0,C 180,E1 24456.574,E2 24456.574} C_VEL
LIN {X 0,Y 517.848,Z 393.088,A -85,B 0,C 180,E1 24453.13,E2 24453.13} C_VEL
LIN {X 0,Y 518.31,Z 381.96,A -85,B 0,C 180,E1 24451.67,E2 24451.67} C_VEL
LIN {X 0,Y 514.494,Z 368.743,A -85,B 0,C 180,E1 24449.484,E2 24449.484} C_VEL
LIN {X 0,Y 512.62,Z 362.947,A -85,B 0,C 180,E1 24448.419,E2 24448.419} C_VEL
LIN {X 0,Y 512.585,Z 362.949,A -85,B 0,C 180,E1 24445.143,E2 24445.143} C_VEL
LIN {X 0,Y 512.572,Z 362.949,A -85,B 0,C 180,E1 24441.661,E2 24441.661} C_VEL
LIN {X 0,Y 512.626,Z 362.946,A -85,B 0,C 180,E1 24438.334,E2 24438.334} C_VEL
LIN {X 0,Y 512.582,Z 362.948,A -85,B 0,C 180,E1 24435.079,E2 24435.079} C_VEL
LIN {X 0,Y 512.576,Z 362.95,A -85,B 0,C 180,E1 24431.66,E2 24431.66} C_VEL
LIN {X 0,Y 512.64,Z 362.945,A -85,B 0,C 180,E1 24428.333,E2 24428.333} C_VEL
LIN {X 0,Y 512.577,Z 362.986,A -85,B 0,C 180,E1 24425.216,E2 24425.216} C_VEL
LIN {X 0,Y 517.488,Z 376.312,A -85,B 0,C 180,E1 24423.413,E2 24423.413} C_VEL
LIN {X 0,Y 520.537,Z 385.915,A -85,B 0,C 180,E1 24422.276,E2 24422.276} C_VEL
LIN {X 0,Y 518.761,Z 420.577,A -85,B 0,C 180,E1 24419.404,E2 24419.404} C_VEL
LIN {X 0,Y 517.266,Z 461.609,A -85,B 0,C 180,E1 24416.21,E2 24416.21} C_VEL
LIN {X 0,Y 519.099,Z 476.93,A -85,B 0,C 180,E1 24415.869,E2 24415.869} C_VEL
LIN {X 0,Y 517.802,Z 620.048,A -85,B 0,C 180,E1 24413.741,E2 24413.741} C_VEL
LIN {X 0,Y 517.463,Z 671.34,A -85,B 0,C 180,E1 24412.999,E2 24412.999} C_VEL
LIN {X 0,Y 517.055,Z 690.393,A -85,B 0,C 180,E1 24412.52,E2 24412.52} C_VEL
LIN {X 0,Y 516.544,Z 708.605,A -85,B 0,C 180,E1 24411.861,E2 24411.861} C_VEL
LIN {X 0,Y 515.961,Z 726.426,A -85,B 0,C 180,E1 24411.008,E2 24411.008} C_VEL
LIN {X 0,Y 515.329,Z 743.661,A -85,B 0,C 180,E1 24409.967,E2 24409.967} C_VEL
LIN {X 0,Y 514.646,Z 760.69,A -85,B 0,C 180,E1 24408.697,E2 24408.697} C_VEL
LIN {X 0,Y 514.031,Z 775.943,A -85,B 0,C 180,E1 24407.314,E2 24407.314} C_VEL
LIN {X 0,Y 513.463,Z 789.691,A -85,B 0,C 180,E1 24405.82,E2 24405.82} C_VEL
LIN {X 0,Y 512.983,Z 802.05,A -85,B 0,C 180,E1 24404.217,E2 24404.217} C_VEL
LIN {X 0,Y 512.619,Z 812.201,A -85,B 0,C 180,E1 24402.618,E2 24402.618} C_VEL
LIN {X 0,Y 512.308,Z 821.476,A -85,B 0,C 180,E1 24400.799,E2 24400.799} C_VEL
LIN {X 0,Y 512.085,Z 829.773,A -85,B 0,C 180,E1 24398.76,E2 24398.76} C_VEL
LIN {X 0,Y 511.973,Z 836.111,A -85,B 0,C 180,E1 24396.729,E2 24396.729} C_VEL
LIN {X 0,Y 511.929,Z 840.668,A -85,B 0,C 180,E1 24394.705,E2 24394.705} C_VEL
LIN {X 0,Y 511.911,Z 843.677,A -85,B 0,C 180,E1 24392.575,E2 24392.575} C_VEL
LIN {X 0,Y 511.908,Z 844.916,A -85,B 0,C 180,E1 24390.448,E2 24390.448} C_VEL
LIN {X 0,Y 511.91,Z 844.414,A -85,B 0,C 180,E1 24388.321,E2 24388.321} C_VEL
LIN {X 0,Y 511.918,Z 842.16,A -85,B 0,C 180,E1 24386.192,E2 24386.192} C_VEL
LIN {X 0,Y 511.946,Z 838.348,A -85,B 0,C 180,E1 24384.171,E2 24384.171} C_VEL
LIN {X 0,Y 512.029,Z 832.818,A -85,B 0,C 180,E1 24382.144,E2 24382.144} C_VEL
LIN {X 0,Y 512.196,Z 825.425,A -85,B 0,C 180,E1 24380.108,E2 24380.108} C_VEL
LIN {X 0,Y 512.473,Z 816.516,A -85,B 0,C 180,E1 24378.179,E2 24378.179} C_VEL
LIN {X 0,Y 512.791,Z 807.401,A -85,B 0,C 180,E1 24376.583,E2 24376.583} C_VEL
LIN {X 0,Y 513.244,Z 795.342,A -85,B 0,C 180,E1 24374.868,E2 24374.868} C_VEL
LIN {X 0,Y 513.819,Z 781.768,A -85,B 0,C 180,E1 24373.262,E2 24373.262} C_VEL
LIN {X 0,Y 514.458,Z 766.567,A -85,B 0,C 180,E1 24371.765,E2 24371.765} C_VEL
LIN {X 0,Y 515.12,Z 751.013,A -85,B 0,C 180,E1 24370.497,E2 24370.497} C_VEL
LIN {X 0,Y 515.77,Z 734.767,A -85,B 0,C 180,E1 24369.405,E2 24369.405} C_VEL
LIN {X 0,Y 516.418,Z 717.101,A -85,B 0,C 180,E1 24368.448,E2 24368.448} C_VEL
LIN {X 0,Y 516.99,Z 699.397,A -85,B 0,C 180,E1 24367.706,E2 24367.706} C_VEL
LIN {X 0,Y 517.479,Z 680.67,A -85,B 0,C 180,E1 24367.132,E2 24367.132} C_VEL
LIN {X 0,Y 517.803,Z 661.043,A -85,B 0,C 180,E1 24366.747,E2 24366.747} C_VEL
LIN {X 0,Y 519.072,Z 474.49,A -85,B 0,C 180,E1 24364.06,E2 24364.06} C_VEL
LIN {X 0,Y 517.446,Z 462.81,A -85,B 0,C 180,E1 24363.798,E2 24363.798} C_VEL
LIN {X 0,Y 519.075,Z 417.817,A -85,B 0,C 180,E1 24360.311,E2 24360.311} C_VEL
LIN {X 0,Y 520.347,Z 385.293,A -85,B 0,C 180,E1 24357.711,E2 24357.711} C_VEL
LIN {X 0,Y 512.598,Z 362.946,A -85,B 0,C 180,E1 24355.241,E2 24355.241} C_VEL
LIN {X 0,Y 512.608,Z 362.948,A -85,B 0,C 180,E1 24351.948,E2 24351.948} C_VEL
LIN {X 0,Y 512.572,Z 362.947,A -85,B 0,C 180,E1 24348.602,E2 24348.602} C_VEL
LIN {X 0,Y 512.609,Z 362.946,A -85,B 0,C 180,E1 24345.234,E2 24345.234} C_VEL
LIN {X 0,Y 512.591,Z 362.948,A -85,B 0,C 180,E1 24341.994,E2 24341.994} C_VEL
LIN {X 0,Y 512.571,Z 362.948,A -85,B 0,C 180,E1 24338.625,E2 24338.625} C_VEL
LIN {X 0,Y 512.623,Z 362.947,A -85,B 0,C 180,E1 24335.264,E2 24335.264} C_VEL
LIN {X 0,Y 512.587,Z 362.953,A -85,B 0,C 180,E1 24331.912,E2 24331.912} C_VEL
LIN {X 0,Y 512.591,Z 363.007,A -85,B 0,C 180,E1 24330.799,E2 24330.799} C_VEL
LIN {X 0,Y 517.716,Z 379.399,A -85,B 0,C 180,E1 24328.969,E2 24328.969} C_VEL
LIN {X 0,Y 518.493,Z 383.251,A -85,B 0,C 180,E1 24328.571,E2 24328.571} C_VEL
LIN {X 0,Y 518.129,Z 408.146,A -85,B 0,C 180,E1 24326.357,E2 24326.357} C_VEL
LIN {X 0,Y 520.025,Z 419.625,A -85,B 0,C 180,E1 24326.046,E2 24326.046} C_VEL
LIN {X 0,Y 518.286,Z 554.871,A -85,B 0,C 180,E1 24323.933,E2 24323.933} C_VEL
LIN {X 0,Y 517.744,Z 616.018,A -85,B 0,C 180,E1 24322.998,E2 24322.998} C_VEL
LIN {X 0,Y 517.372,Z 635.328,A -85,B 0,C 180,E1 24322.49,E2 24322.49} C_VEL
LIN {X 0,Y 516.852,Z 653.811,A -85,B 0,C 180,E1 24321.786,E2 24321.786} C_VEL
LIN {X 0,Y 516.255,Z 670.782,A -85,B 0,C 180,E1 24320.936,E2 24320.936} C_VEL
LIN {X 0,Y 515.583,Z 687.337,A -85,B 0,C 180,E1 24319.892,E2 24319.892} C_VEL
LIN {X 0,Y 514.898,Z 702.854,A -85,B 0,C 180,E1 24318.687,E2 24318.687} C_VEL
LIN {X 0,Y 514.207,Z 717.529,A -85,B 0,C 180,E1 24317.304,E2 24317.304} C_VEL
LIN {X 0,Y 513.59,Z 730.641,A -85,B 0,C 180,E1 24315.816,E2 24315.816} C_VEL
LIN {X 0,Y 513.026,Z 743.173,A -85,B 0,C 180,E1 24314.1,E2 24314.1} C_VEL
LIN {X 0,Y 512.585,Z 754.068,A -85,B 0,C 180,E1 24312.276,E2 24312.276} C_VEL
LIN {X 0,Y 512.261,Z 763.406,A -85,B 0,C 180,E1 24310.345,E2 24310.345} C_VEL
LIN {X 0,Y 512.07,Z 770.835,A -85,B 0,C 180,E1 24308.421,E2 24308.421} C_VEL
LIN {X 0,Y 511.966,Z 776.581,A -85,B 0,C 180,E1 24306.504,E2 24306.504} C_VEL
LIN {X 0,Y 511.922,Z 780.98,A -85,B 0,C 180,E1 24304.481,E2 24304.481} C_VEL
LIN {X 0,Y 511.909,Z 783.786,A -85,B 0,C 180,E1 24302.463,E2 24302.463} C_VEL
LIN {X 0,Y 511.908,Z 784.893,A -85,B 0,C 180,E1 24300.448,E2 24300.448} C_VEL
LIN {X 0,Y 511.909,Z 784.435,A -85,B 0,C 180,E1 24298.321,E2 24298.321} C_VEL
LIN {X 0,Y 511.914,Z 782.419,A -85,B 0,C 180,E1 24296.304,E2 24296.304} C_VEL
LIN {X 0,Y 511.941,Z 778.685,A -85,B 0,C 180,E1 24294.283,E2 24294.283} C_VEL
LIN {X 0,Y 512.021,Z 773.313,A -85,B 0,C 180,E1 24292.256,E2 24292.256} C_VEL
LIN {X 0,Y 512.179,Z 766.163,A -85,B 0,C 180,E1 24290.221,E2 24290.221} C_VEL
LIN {X 0,Y 512.452,Z 757.45,A -85,B 0,C 180,E1 24288.292,E2 24288.292} C_VEL
LIN {X 0,Y 512.843,Z 747.307,A -85,B 0,C 180,E1 24286.47,E2 24286.47} C_VEL
LIN {X 0,Y 513.351,Z 735.733,A -85,B 0,C 180,E1 24284.755,E2 24284.755} C_VEL
LIN {X 0,Y 513.97,Z 722.602,A -85,B 0,C 180,E1 24283.15,E2 24283.15} C_VEL
LIN {X 0,Y 514.687,Z 707.88,A -85,B 0,C 180,E1 24281.657,E2 24281.657} C_VEL
LIN {X 0,Y 515.428,Z 692.144,A -85,B 0,C 180,E1 24280.347,E2 24280.347} C_VEL
LIN {X 0,Y 516.139,Z 675.794,A -85,B 0,C 180,E1 24279.237,E2 24279.237} C_VEL
LIN {X 0,Y 516.805,Z 658.858,A -85,B 0,C 180,E1 24278.313,E2 24278.313} C_VEL
LIN {X 0,Y 517.397,Z 640.668,A -85,B 0,C 180,E1 24277.548,E2 24277.548} C_VEL
LIN {X 0,Y 517.868,Z 622.026,A -85,B 0,C 180,E1 24276.981,E2 24276.981} C_VEL
LIN {X 0,Y 518.179,Z 601.61,A -85,B 0,C 180,E1 24276.586,E2 24276.586} C_VEL
LIN {X 0,Y 519.493,Z 467.04,A -85,B 0,C 180,E1 24274.58,E2 24274.58} C_VEL
LIN {X 0,Y 518.673,Z 459.457,A -85,B 0,C 180,E1 24274.42,E2 24274.42} C_VEL
LIN {X 0,Y 513.284,Z 439.638,A -85,B 0,C 180,E1 24273.816,E2 24273.816} C_VEL
LIN {X 0,Y 512.673,Z 433.126,A -85,B 0,C 180,E1 24273.676,E2 24273.676} C_VEL
LIN {X 0,Y 512.675,Z 418.457,A -85,B 0,C 180,E1 24273.427,E2 24273.427} C_VEL
LIN {X 0,Y 510.303,Z 405.655,A -85,B 0,C 180,E1 24273.063,E2 24273.063} C_VEL
LIN {X 0,Y 510.812,Z 384.145,A -85,B 0,C 180,E1 24271.04,E2 24271.04} C_VEL
LIN {X 0,Y 504.698,Z 363.933,A -85,B 0,C 180,E1 24268.685,E2 24268.685} C_VEL
LIN {X 0,Y 504.641,Z 363.936,A -85,B 0,C 180,E1 24265.311,E2 24265.311} C_VEL
LIN {X 0,Y 504.642,Z 363.936,A -85,B 0,C 180,E1 24261.817,E2 24261.817} C_VEL
LIN {X 0,Y 504.703,Z 363.933,A -85,B 0,C 180,E1 24258.491,E2 24258.491} C_VEL
LIN {X 0,Y 504.642,Z 363.934,A -85,B 0,C 180,E1 24255.142,E2 24255.142} C_VEL
LIN {X 0,Y 504.637,Z 363.933,A -85,B 0,C 180,E1 24251.587,E2 24251.587} C_VEL
LIN {X 0,Y 504.7,Z 363.933,A -85,B 0,C 180,E1 24248.322,E2 24248.322} C_VEL
LIN {X 0,Y 504.649,Z 363.934,A -85,B 0,C 180,E1 24244.889,E2 24244.889} C_VEL
LIN {X 0,Y 504.635,Z 363.934,A -85,B 0,C 180,E1 24241.406,E2 24241.406} C_VEL
LIN {X 0,Y 504.692,Z 363.934,A -85,B 0,C 180,E1 24238.132,E2 24238.132} C_VEL
LIN {X 0,Y 504.655,Z 363.933,A -85,B 0,C 180,E1 24234.712,E2 24234.712} C_VEL
LIN {X 0,Y 504.634,Z 363.932,A -85,B 0,C 180,E1 24231.259,E2 24231.259} C_VEL
LIN {X 0,Y 504.676,Z 363.932,A -85,B 0,C 180,E1 24227.884,E2 24227.884} C_VEL
LIN {X 0,Y 504.655,Z 363.934,A -85,B 0,C 180,E1 24224.574,E2 24224.574} C_VEL
LIN {X 0,Y 504.634,Z 363.934,A -85,B 0,C 180,E1 24221.196,E2 24221.196} C_VEL
LIN {X 0,Y 504.683,Z 363.934,A -85,B 0,C 180,E1 24217.857,E2 24217.857} C_VEL
LIN {X 0,Y 504.649,Z 363.932,A -85,B 0,C 180,E1 24214.546,E2 24214.546} C_VEL
LIN {X 0,Y 504.633,Z 363.934,A -85,B 0,C 180,E1 24211.135,E2 24211.135} C_VEL
LIN {X 0,Y 504.69,Z 363.931,A -85,B 0,C 180,E1 24207.843,E2 24207.843} C_VEL
LIN {X 0,Y 504.65,Z 363.933,A -85,B 0,C 180,E1 24204.429,E2 24204.429} C_VEL
LIN {X 0,Y 504.633,Z 363.933,A -85,B 0,C 180,E1 24200.995,E2 24200.995} C_VEL
LIN {X 0,Y 504.679,Z 363.934,A -85,B 0,C 180,E1 24197.614,E2 24197.614} C_VEL
LIN {X 0,Y 504.647,Z 363.934,A -85,B 0,C 180,E1 24194.348,E2 24194.348} C_VEL
LIN {X 0,Y 504.635,Z 363.934,A -85,B 0,C 180,E1 24190.918,E2 24190.918} C_VEL
LIN {X 0,Y 504.682,Z 363.934,A -85,B 0,C 180,E1 24187.52,E2 24187.52} C_VEL
LIN {X 0,Y 504.659,Z 363.933,A -85,B 0,C 180,E1 24184.092,E2 24184.092} C_VEL
LIN {X 0,Y 504.63,Z 363.933,A -85,B 0,C 180,E1 24180.669,E2 24180.669} C_VEL
LIN {X 0,Y 504.673,Z 363.936,A -85,B 0,C 180,E1 24177.354,E2 24177.354} C_VEL
LIN {X 0,Y 504.661,Z 363.936,A -85,B 0,C 180,E1 24173.935,E2 24173.935} C_VEL
LIN {X 0,Y 504.631,Z 363.935,A -85,B 0,C 180,E1 24170.6,E2 24170.6} C_VEL
LIN {X 0,Y 504.68,Z 363.935,A -85,B 0,C 180,E1 24167.309,E2 24167.309} C_VEL
LIN {X 0,Y 504.655,Z 363.934,A -85,B 0,C 180,E1 24163.904,E2 24163.904} C_VEL
LIN {X 0,Y 504.631,Z 363.936,A -85,B 0,C 180,E1 24160.533,E2 24160.533} C_VEL
LIN {X 0,Y 504.677,Z 363.937,A -85,B 0,C 180,E1 24157.176,E2 24157.176} C_VEL
LIN {X 0,Y 504.651,Z 363.937,A -85,B 0,C 180,E1 24153.831,E2 24153.831} C_VEL
LIN {X 0,Y 504.642,Z 363.998,A -85,B 0,C 180,E1 24150.575,E2 24150.575} C_VEL
LIN {X 0,Y 509.266,Z 381.724,A -85,B 0,C 180,E1 24147.985,E2 24147.985} C_VEL
LIN {X 0,Y 508.15,Z 409.475,A -85,B 0,C 180,E1 24144.53,E2 24144.53} C_VEL
LIN {X 0,Y 507.165,Z 438.07,A -85,B 0,C 180,E1 24141.027,E2 24141.027} C_VEL
LIN {X 0,Y 506.224,Z 467.73,A -85,B 0,C 180,E1 24137.447,E2 24137.447} C_VEL
LIN {X 0,Y 505.948,Z 480.463,A -85,B 0,C 180,E1 24135.964,E2 24135.964} C_VEL
LIN {X 0,Y 507.582,Z 493.007,A -85,B 0,C 180,E1 24135.699,E2 24135.699} C_VEL
LIN {X 0,Y 506.587,Z 595.826,A -85,B 0,C 180,E1 24134.077,E2 24134.077} C_VEL
LIN {X 0,Y 506.401,Z 610.42,A -85,B 0,C 180,E1 24133.648,E2 24133.648} C_VEL
LIN {X 0,Y 506.105,Z 625.79,A -85,B 0,C 180,E1 24132.958,E2 24132.958} C_VEL
LIN {X 0,Y 505.711,Z 639.608,A -85,B 0,C 180,E1 24132.098,E2 24132.098} C_VEL
LIN {X 0,Y 505.383,Z 651.043,A -85,B 0,C 180,E1 24131.18,E2 24131.18} C_VEL
LIN {X 0,Y 505.034,Z 663.32,A -85,B 0,C 180,E1 24129.918,E2 24129.918} C_VEL
LIN {X 0,Y 504.727,Z 673.661,A -85,B 0,C 180,E1 24128.544,E2 24128.544} C_VEL
LIN {X 0,Y 504.515,Z 681.718,A -85,B 0,C 180,E1 24127.173,E2 24127.173} C_VEL
LIN {X 0,Y 504.355,Z 688.881,A -85,B 0,C 180,E1 24125.575,E2 24125.575} C_VEL
LIN {X 0,Y 504.263,Z 694.287,A -85,B 0,C 180,E1 24123.866,E2 24123.866} C_VEL
LIN {X 0,Y 504.22,Z 697.677,A -85,B 0,C 180,E1 24122.159,E2 24122.159} C_VEL
LIN {X 0,Y 504.229,Z 699.217,A -85,B 0,C 180,E1 24120.455,E2 24120.455} C_VEL
LIN {X 0,Y 504.238,Z 698.988,A -85,B 0,C 180,E1 24118.75,E2 24118.75} C_VEL
LIN {X 0,Y 504.294,Z 696.905,A -85,B 0,C 180,E1 24117.045,E2 24117.045} C_VEL
LIN {X 0,Y 504.375,Z 693.28,A -85,B 0,C 180,E1 24115.452,E2 24115.452} C_VEL
LIN {X 0,Y 504.541,Z 687.347,A -85,B 0,C 180,E1 24113.743,E2 24113.743} C_VEL
LIN {X 0,Y 504.751,Z 679.57,A -85,B 0,C 180,E1 24112.144,E2 24112.144} C_VEL
LIN {X 0,Y 505.025,Z 670.786,A -85,B 0,C 180,E1 24110.772,E2 24110.772} C_VEL
LIN {X 0,Y 505.369,Z 660.534,A -85,B 0,C 180,E1 24109.513,E2 24109.513} C_VEL
LIN {X 0,Y 505.744,Z 647.921,A -85,B 0,C 180,E1 24108.309,E2 24108.309} C_VEL
LIN {X 0,Y 506.149,Z 634.52,A -85,B 0,C 180,E1 24107.334,E2 24107.334} C_VEL
LIN {X 0,Y 506.487,Z 620.954,A -85,B 0,C 180,E1 24106.588,E2 24106.588} C_VEL
LIN {X 0,Y 506.774,Z 606.047,A -85,B 0,C 180,E1 24105.999,E2 24105.999} C_VEL
LIN {X 0,Y 506.97,Z 589.709,A -85,B 0,C 180,E1 24105.602,E2 24105.602} C_VEL
LIN {X 0,Y 508.525,Z 490.627,A -85,B 0,C 180,E1 24103.841,E2 24103.841} C_VEL
LIN {X 0,Y 506.581,Z 480.051,A -85,B 0,C 180,E1 24103.517,E2 24103.517} C_VEL
LIN {X 0,Y 507.753,Z 449.671,A -85,B 0,C 180,E1 24099.782,E2 24099.782} C_VEL
LIN {X 0,Y 509.185,Z 420.267,A -85,B 0,C 180,E1 24096.078,E2 24096.078} C_VEL
LIN {X 0,Y 510.712,Z 393.468,A -85,B 0,C 180,E1 24092.608,E2 24092.608} C_VEL
LIN {X 0,Y 511.064,Z 384.911,A -85,B 0,C 180,E1 24091.455,E2 24091.455} C_VEL
LIN {X 0,Y 507.643,Z 372.869,A -85,B 0,C 180,E1 24089.398,E2 24089.398} C_VEL
LIN {X 0,Y 504.633,Z 363.941,A -85,B 0,C 180,E1 24087.709,E2 24087.709} C_VEL
LIN {X 0,Y 504.674,Z 363.937,A -85,B 0,C 180,E1 24084.321,E2 24084.321} C_VEL
LIN {X 0,Y 504.659,Z 363.937,A -85,B 0,C 180,E1 24080.947,E2 24080.947} C_VEL
LIN {X 0,Y 504.634,Z 363.937,A -85,B 0,C 180,E1 24077.65,E2 24077.65} C_VEL
LIN {X 0,Y 504.679,Z 363.936,A -85,B 0,C 180,E1 24074.217,E2 24074.217} C_VEL
LIN {X 0,Y 504.663,Z 363.937,A -85,B 0,C 180,E1 24070.814,E2 24070.814} C_VEL
LIN {X 0,Y 504.635,Z 363.94,A -85,B 0,C 180,E1 24067.465,E2 24067.465} C_VEL
LIN {X 0,Y 504.669,Z 363.999,A -85,B 0,C 180,E1 24065.94,E2 24065.94} C_VEL
LIN {X 0,Y 509.572,Z 376.884,A -85,B 0,C 180,E1 24064.039,E2 24064.039} C_VEL
LIN {X 0,Y 513.396,Z 388.759,A -85,B 0,C 180,E1 24062.548,E2 24062.548} C_VEL
LIN {X 0,Y 511.358,Z 422.774,A -85,B 0,C 180,E1 24059.65,E2 24059.65} C_VEL
LIN {X 0,Y 509.772,Z 460.555,A -85,B 0,C 180,E1 24056.639,E2 24056.639} C_VEL
LIN {X 0,Y 511.857,Z 477.969,A -85,B 0,C 180,E1 24056.236,E2 24056.236} C_VEL
LIN {X 0,Y 509.773,Z 671.702,A -85,B 0,C 180,E1 24053.242,E2 24053.242} C_VEL
LIN {X 0,Y 509.315,Z 690.473,A -85,B 0,C 180,E1 24052.748,E2 24052.748} C_VEL
LIN {X 0,Y 508.741,Z 709.188,A -85,B 0,C 180,E1 24052.048,E2 24052.048} C_VEL
LIN {X 0,Y 508.077,Z 727.765,A -85,B 0,C 180,E1 24051.125,E2 24051.125} C_VEL
LIN {X 0,Y 507.399,Z 744.809,A -85,B 0,C 180,E1 24050.052,E2 24050.052} C_VEL
LIN {X 0,Y 506.719,Z 760.777,A -85,B 0,C 180,E1 24048.822,E2 24048.822} C_VEL
LIN {X 0,Y 506.062,Z 776.135,A -85,B 0,C 180,E1 24047.39,E2 24047.39} C_VEL
LIN {X 0,Y 505.443,Z 790.45,A -85,B 0,C 180,E1 24045.783,E2 24045.783} C_VEL
LIN {X 0,Y 504.952,Z 802.93,A -85,B 0,C 180,E1 24044.096,E2 24044.096} C_VEL
LIN {X 0,Y 504.55,Z 814.265,A -85,B 0,C 180,E1 24042.242,E2 24042.242} C_VEL
LIN {X 0,Y 504.242,Z 823.973,A -85,B 0,C 180,E1 24040.28,E2 24040.28} C_VEL
LIN {X 0,Y 504.064,Z 831.628,A -85,B 0,C 180,E1 24038.326,E2 24038.326} C_VEL
LIN {X 0,Y 503.966,Z 837.318,A -85,B 0,C 180,E1 24036.379,E2 24036.379} C_VEL
LIN {X 0,Y 503.92,Z 841.678,A -85,B 0,C 180,E1 24034.21,E2 24034.21} C_VEL
LIN {X 0,Y 503.911,Z 844.208,A -85,B 0,C 180,E1 24032.047,E2 24032.047} C_VEL
LIN {X 0,Y 503.914,Z 844.984,A -85,B 0,C 180,E1 24029.886,E2 24029.886} C_VEL
LIN {X 0,Y 503.911,Z 844.018,A -85,B 0,C 180,E1 24027.726,E2 24027.726} C_VEL
LIN {X 0,Y 503.92,Z 841.494,A -85,B 0,C 180,E1 24025.676,E2 24025.676} C_VEL
LIN {X 0,Y 503.966,Z 837.314,A -85,B 0,C 180,E1 24023.621,E2 24023.621} C_VEL
LIN {X 0,Y 504.064,Z 831.627,A -85,B 0,C 180,E1 24021.674,E2 24021.674} C_VEL
LIN {X 0,Y 504.244,Z 824.006,A -85,B 0,C 180,E1 24019.72,E2 24019.72} C_VEL
LIN {X 0,Y 504.549,Z 814.381,A -85,B 0,C 180,E1 24017.758,E2 24017.758} C_VEL
LIN {X 0,Y 504.95,Z 803.168,A -85,B 0,C 180,E1 24015.904,E2 24015.904} C_VEL
LIN {X 0,Y 505.476,Z 790.378,A -85,B 0,C 180,E1 24014.159,E2 24014.159} C_VEL
LIN {X 0,Y 506.091,Z 776.668,A -85,B 0,C 180,E1 24012.6,E2 24012.6} C_VEL
LIN {X 0,Y 506.768,Z 761.711,A -85,B 0,C 180,E1 24011.18,E2 24011.18} C_VEL
LIN {X 0,Y 507.472,Z 746.108,A -85,B 0,C 180,E1 24009.951,E2 24009.951} C_VEL
LIN {X 0,Y 508.171,Z 729.826,A -85,B 0,C 180,E1 24008.896,E2 24008.896} C_VEL
LIN {X 0,Y 508.856,Z 712.371,A -85,B 0,C 180,E1 24007.99,E2 24007.99} C_VEL
LIN {X 0,Y 509.474,Z 694.005,A -85,B 0,C 180,E1 24007.263,E2 24007.263} C_VEL
LIN {X 0,Y 509.955,Z 675.141,A -85,B 0,C 180,E1 24006.733,E2 24006.733} C_VEL
LIN {X 0,Y 510.277,Z 650.389,A -85,B 0,C 180,E1 24006.314,E2 24006.314} C_VEL
LIN {X 0,Y 511.584,Z 475.215,A -85,B 0,C 180,E1 24003.738,E2 24003.738} C_VEL
LIN {X 0,Y 509.947,Z 462.054,A -85,B 0,C 180,E1 24003.391,E2 24003.391} C_VEL
LIN {X 0,Y 511.77,Z 417.408,A -85,B 0,C 180,E1 23999.86,E2 23999.86} C_VEL
LIN {X 0,Y 513.029,Z 387.98,A -85,B 0,C 180,E1 23997.459,E2 23997.459} C_VEL
LIN {X 0,Y 505.283,Z 366.224,A -85,B 0,C 180,E1 23995.007,E2 23995.007} C_VEL
LIN {X 0,Y 504.633,Z 363.936,A -85,B 0,C 180,E1 23994.718,E2 23994.718} C_VEL
LIN {X 0,Y 504.672,Z 363.933,A -85,B 0,C 180,E1 23991.315,E2 23991.315} C_VEL
LIN {X 0,Y 504.663,Z 363.937,A -85,B 0,C 180,E1 23987.959,E2 23987.959} C_VEL
LIN {X 0,Y 504.632,Z 363.937,A -85,B 0,C 180,E1 23984.54,E2 23984.54} C_VEL
LIN {X 0,Y 504.663,Z 363.936,A -85,B 0,C 180,E1 23981.13,E2 23981.13} C_VEL
LIN {X 0,Y 504.654,Z 363.937,A -85,B 0,C 180,E1 23977.893,E2 23977.893} C_VEL
LIN {X 0,Y 504.632,Z 363.939,A -85,B 0,C 180,E1 23974.487,E2 23974.487} C_VEL
LIN {X 0,Y 504.701,Z 363.984,A -85,B 0,C 180,E1 23971.314,E2 23971.314} C_VEL
LIN {X 0,Y 510.087,Z 380.707,A -85,B 0,C 180,E1 23969.389,E2 23969.389} C_VEL
LIN {X 0,Y 511.285,Z 385.975,A -85,B 0,C 180,E1 23968.824,E2 23968.824} C_VEL
LIN {X 0,Y 510.946,Z 409.1,A -85,B 0,C 180,E1 23966.766,E2 23966.766} C_VEL
LIN {X 0,Y 512.871,Z 420.851,A -85,B 0,C 180,E1 23966.43,E2 23966.43} C_VEL
LIN {X 0,Y 510.877,Z 549.933,A -85,B 0,C 180,E1 23964.332,E2 23964.332} C_VEL
LIN {X 0,Y 510.192,Z 616.874,A -85,B 0,C 180,E1 23963.282,E2 23963.282} C_VEL
LIN {X 0,Y 509.792,Z 636.167,A -85,B 0,C 180,E1 23962.763,E2 23962.763} C_VEL
LIN {X 0,Y 509.265,Z 654.046,A -85,B 0,C 180,E1 23962.074,E2 23962.074} C_VEL
LIN {X 0,Y 508.625,Z 671.215,A -85,B 0,C 180,E1 23961.205,E2 23961.205} C_VEL
LIN {X 0,Y 507.913,Z 687.748,A -85,B 0,C 180,E1 23960.151,E2 23960.151} C_VEL
LIN {X 0,Y 507.178,Z 703.387,A -85,B 0,C 180,E1 23958.923,E2 23958.923} C_VEL
LIN {X 0,Y 506.44,Z 718.029,A -85,B 0,C 180,E1 23957.525,E2 23957.525} C_VEL
LIN {X 0,Y 505.747,Z 731.673,A -85,B 0,C 180,E1 23955.95,E2 23955.95} C_VEL
LIN {X 0,Y 505.142,Z 744.134,A -85,B 0,C 180,E1 23954.208,E2 23954.208} C_VEL
LIN {X 0,Y 504.67,Z 754.994,A -85,B 0,C 180,E1 23952.355,E2 23952.355} C_VEL
LIN {X 0,Y 504.322,Z 764.293,A -85,B 0,C 180,E1 23950.394,E2 23950.394} C_VEL
LIN {X 0,Y 504.099,Z 771.993,A -85,B 0,C 180,E1 23948.325,E2 23948.325} C_VEL
LIN {X 0,Y 503.98,Z 777.79,A -85,B 0,C 180,E1 23946.264,E2 23946.264} C_VEL
LIN {X 0,Y 503.924,Z 781.791,A -85,B 0,C 180,E1 23944.21,E2 23944.21} C_VEL
LIN {X 0,Y 503.913,Z 784.307,A -85,B 0,C 180,E1 23942.047,E2 23942.047} C_VEL
LIN {X 0,Y 503.92,Z 785.14,A -85,B 0,C 180,E1 23939.886,E2 23939.886} C_VEL
LIN {X 0,Y 503.913,Z 784.202,A -85,B 0,C 180,E1 23937.726,E2 23937.726} C_VEL
LIN {X 0,Y 503.929,Z 781.542,A -85,B 0,C 180,E1 23935.562,E2 23935.562} C_VEL
LIN {X 0,Y 503.985,Z 777.39,A -85,B 0,C 180,E1 23933.507,E2 23933.507} C_VEL
LIN {X 0,Y 504.106,Z 771.478,A -85,B 0,C 180,E1 23931.445,E2 23931.445} C_VEL
LIN {X 0,Y 504.33,Z 763.596,A -85,B 0,C 180,E1 23929.375,E2 23929.375} C_VEL
LIN {X 0,Y 504.681,Z 754.117,A -85,B 0,C 180,E1 23927.412,E2 23927.412} C_VEL
LIN {X 0,Y 505.174,Z 743.095,A -85,B 0,C 180,E1 23925.559,E2 23925.559} C_VEL
LIN {X 0,Y 505.762,Z 731.16,A -85,B 0,C 180,E1 23923.904,E2 23923.904} C_VEL
LIN {X 0,Y 506.486,Z 717.245,A -85,B 0,C 180,E1 23922.301,E2 23922.301} C_VEL
LIN {X 0,Y 507.25,Z 702.554,A -85,B 0,C 180,E1 23920.9,E2 23920.9} C_VEL
LIN {X 0,Y 508.015,Z 687.044,A -85,B 0,C 180,E1 23919.679,E2 23919.679} C_VEL
LIN {X 0,Y 508.776,Z 670.541,A -85,B 0,C 180,E1 23918.62,E2 23918.62} C_VEL
LIN {X 0,Y 509.48,Z 653.353,A -85,B 0,C 180,E1 23917.743,E2 23917.743} C_VEL
LIN {X 0,Y 510.098,Z 634.429,A -85,B 0,C 180,E1 23917.009,E2 23917.009} C_VEL
LIN {X 0,Y 510.545,Z 615.253,A -85,B 0,C 180,E1 23916.498,E2 23916.498} C_VEL
LIN {X 0,Y 511.057,Z 566.553,A -85,B 0,C 180,E1 23915.732,E2 23915.732} C_VEL
LIN {X 0,Y 512.673,Z 433.126,A -85,B 0,C 180,E1 23913.676,E2 23913.676} C_VEL
LIN {X 0,Y 511.768,Z 428.185,A -85,B 0,C 180,E1 23913.542,E2 23913.542} C_VEL
LIN {X 0,Y 507.793,Z 420.627,A -85,B 0,C 180,E1 23913.192,E2 23913.192} C_VEL
LIN {X 0,Y 504.602,Z 414.156,A -85,B 0,C 180,E1 23912.899,E2 23912.899} C_VEL
LIN {X 0,Y 504.059,Z 412.019,A -85,B 0,C 180,E1 23912.83,E2 23912.83} C_VEL
LIN {X 0,Y 502.938,Z 406.134,A -85,B 0,C 180,E1 23912.662,E2 23912.662} C_VEL
LIN {X 0,Y 503.399,Z 386.685,A -85,B 0,C 180,E1 23910.816,E2 23910.816} C_VEL
LIN {X 0,Y 497.535,Z 367.496,A -85,B 0,C 180,E1 23908.55,E2 23908.55} C_VEL
LIN {X 0,Y 496.73,Z 364.924,A -85,B 0,C 180,E1 23908.239,E2 23908.239} C_VEL
LIN {X 0,Y 496.74,Z 364.924,A -85,B 0,C 180,E1 23904.807,E2 23904.807} C_VEL
LIN {X 0,Y 496.7,Z 364.924,A -85,B 0,C 180,E1 23901.357,E2 23901.357} C_VEL
LIN {X 0,Y 496.702,Z 364.924,A -85,B 0,C 180,E1 23897.752,E2 23897.752} C_VEL
LIN {X 0,Y 496.756,Z 364.923,A -85,B 0,C 180,E1 23894.394,E2 23894.394} C_VEL
LIN {X 0,Y 496.709,Z 364.922,A -85,B 0,C 180,E1 23890.986,E2 23890.986} C_VEL
LIN {X 0,Y 496.699,Z 364.923,A -85,B 0,C 180,E1 23887.521,E2 23887.521} C_VEL
LIN {X 0,Y 496.748,Z 364.924,A -85,B 0,C 180,E1 23884.165,E2 23884.165} C_VEL
LIN {X 0,Y 496.721,Z 364.922,A -85,B 0,C 180,E1 23880.737,E2 23880.737} C_VEL
LIN {X 0,Y 496.697,Z 364.922,A -85,B 0,C 180,E1 23877.321,E2 23877.321} C_VEL
LIN {X 0,Y 496.728,Z 364.922,A -85,B 0,C 180,E1 23873.866,E2 23873.866} C_VEL
LIN {X 0,Y 496.731,Z 364.921,A -85,B 0,C 180,E1 23870.502,E2 23870.502} C_VEL
LIN {X 0,Y 496.696,Z 364.92,A -85,B 0,C 180,E1 23867.092,E2 23867.092} C_VEL
LIN {X 0,Y 496.716,Z 364.921,A -85,B 0,C 180,E1 23863.622,E2 23863.622} C_VEL
